   LaserStart_Ext()
   LIN {X 1.720, Y -28.438, Z 22.950}
   LaserEnd_Ext()
   LIN {X 2.720, Y -27.441, Z 22.950}
   LaserStart_Ext()
   LIN {X 2.720, Y 39.118, Z 22.950}
   LaserEnd_Ext()
   LIN {X 3.720, Y 35.905, Z 22.950}
   LaserStart_Ext()
   LIN {X 3.720, Y -25.441, Z 22.950}
   LaserEnd_Ext()
   LIN {X 4.720, Y -22.355, Z 22.950}
   LaserStart_Ext()
   LIN {X 4.720, Y 32.224, Z 22.950}
   LaserEnd_Ext()
   LIN {X 5.720, Y 28.019, Z 22.950}
   LaserStart_Ext()
   LIN {X 5.720, Y -18.121, Z 22.950}
   LaserEnd_Ext()
   LIN {X 6.720, Y -12.774, Z 22.950}
   LaserStart_Ext()
   LIN {X 6.720, Y 22.583, Z 22.950}
   LaserEnd_Ext()
   LIN {X 7.720, Y 14.905, Z 22.950}
   LaserStart_Ext()
   LIN {X 7.720, Y -4.969, Z 22.950}
   LaserEnd_Ext()
   LIN {X -0.569, Y -18.768, Z 23.800}
   LaserStart_Ext()
   LIN {X 0.218, Y -19.359, Z 23.800} C_DIS
   LIN {X 0.697, Y -20.340, Z 23.800} C_DIS
   LIN {X 1.338, Y -21.643, Z 23.800} C_DIS
   LIN {X 1.314, Y -22.747, Z 23.800} C_DIS
   LIN {X 1.286, Y -23.819, Z 23.800} C_DIS
   LIN {X 0.696, Y -24.975, Z 23.800} C_DIS
   LIN {X 0.224, Y -25.880, Z 23.800} C_DIS
   LIN {X -0.464, Y -26.392, Z 23.800} C_DIS
   LIN {X -1.551, Y -27.214, Z 23.800} C_DIS
   LIN {X -3.664, Y -27.649, Z 23.800} C_DIS
   LIN {X -3.922, Y -27.593, Z 23.800} C_DIS
   LIN {X -5.673, Y -27.207, Z 23.800} C_DIS
   LIN {X -7.126, Y -26.129, Z 23.800} C_DIS
   LIN {X -7.331, Y -25.976, Z 23.800} C_DIS
   LIN {X -7.494, Y -25.689, Z 23.800} C_DIS
   LIN {X -8.349, Y -24.188, Z 23.800} C_DIS
   LIN {X -8.499, Y -22.630, Z 23.800} C_DIS
   LIN {X -8.549, Y -22.171, Z 23.800} C_DIS
   LIN {X -8.508, Y -21.998, Z 23.800} C_DIS
   LIN {X -8.307, Y -21.606, Z 23.800} C_DIS
   LIN {X -7.236, Y -19.264, Z 23.800} C_DIS
   LIN {X -5.530, Y -18.053, Z 23.800} C_DIS
   LIN {X -4.970, Y -17.940, Z 23.800} C_DIS
   LIN {X -3.503, Y -17.647, Z 23.800} C_DIS
   LIN {X -2.373, Y -17.894, Z 23.800} C_DIS
   LIN {X -1.482, Y -18.086, Z 23.800} C_DIS
   LIN {X -0.569, Y -18.768, Z 23.800}
   LaserEnd_Ext()
   LIN {X -9.493, Y -14.716, Z 23.800}
   LaserStart_Ext()
   LIN {X -9.270, Y -14.247, Z 23.800} C_DIS
   LIN {X -7.563, Y -10.615, Z 23.800} C_DIS
   LIN {X -6.096, Y -6.905, Z 23.800} C_DIS
   LIN {X -5.884, Y -6.373, Z 23.800} C_DIS
   LIN {X -5.593, Y -5.440, Z 23.800} C_DIS
   LIN {X -4.023, Y -0.432, Z 23.800} C_DIS
   LIN {X -3.188, Y 3.138, Z 23.800} C_DIS
   LIN {X -2.971, Y 4.113, Z 23.800} C_DIS
   LIN {X -2.513, Y 6.884, Z 23.800} C_DIS
   LIN {X -2.208, Y 8.691, Z 23.800} C_DIS
   LIN {X -2.174, Y 8.967, Z 23.800} C_DIS
   LIN {X -1.817, Y 12.348, Z 23.800} C_DIS
   LIN {X -1.729, Y 13.559, Z 23.800} C_DIS
   LIN {X -1.697, Y 15.626, Z 23.800} C_DIS
   LIN {X -1.672, Y 18.321, Z 23.800} C_DIS
   LIN {X -1.649, Y 21.542, Z 23.800} C_DIS
   LIN {X -1.905, Y 24.867, Z 23.800} C_DIS
   LIN {X -2.060, Y 26.694, Z 23.800} C_DIS
   LIN {X -2.450, Y 29.467, Z 23.800} C_DIS
   LIN {X -2.582, Y 30.379, Z 23.800} C_DIS
   LIN {X -3.012, Y 32.709, Z 23.800} C_DIS
   LIN {X -3.518, Y 35.029, Z 23.800} C_DIS
   LIN {X -3.817, Y 36.241, Z 23.800} C_DIS
   LIN {X -3.902, Y 36.583, Z 23.800} C_DIS
   LIN {X -4.015, Y 37.014, Z 23.800} C_DIS
   LIN {X -4.218, Y 37.794, Z 23.800} C_DIS
   LIN {X -4.291, Y 38.488, Z 23.800} C_DIS
   LIN {X -4.358, Y 39.188, Z 23.800} C_DIS
   LIN {X -4.077, Y 40.123, Z 23.800} C_DIS
   LIN {X -3.903, Y 40.742, Z 23.800} C_DIS
   LIN {X -3.579, Y 41.112, Z 23.800} C_DIS
   LIN {X -2.716, Y 42.095, Z 23.800} C_DIS
   LIN {X -0.784, Y 42.721, Z 23.800} C_DIS
   LIN {X -0.398, Y 42.840, Z 23.800} C_DIS
   LIN {X -0.004, Y 42.750, Z 23.800} C_DIS
   LIN {X 1.306, Y 42.455, Z 23.800} C_DIS
   LIN {X 1.975, Y 41.937, Z 23.800} C_DIS
   LIN {X 2.681, Y 41.387, Z 23.800} C_DIS
   LIN {X 3.233, Y 40.398, Z 23.800} C_DIS
   LIN {X 3.399, Y 40.101, Z 23.800} C_DIS
   LIN {X 3.476, Y 39.867, Z 23.800} C_DIS
   LIN {X 3.864, Y 38.690, Z 23.800} C_DIS
   LIN {X 4.445, Y 36.821, Z 23.800} C_DIS
   LIN {X 4.562, Y 36.440, Z 23.800} C_DIS
   LIN {X 4.847, Y 35.435, Z 23.800} C_DIS
   LIN {X 5.308, Y 33.824, Z 23.800} C_DIS
   LIN {X 5.446, Y 33.304, Z 23.800} C_DIS
   LIN {X 6.101, Y 30.733, Z 23.800} C_DIS
   LIN {X 6.906, Y 27.137, Z 23.800} C_DIS
   LIN {X 6.995, Y 26.718, Z 23.800} C_DIS
   LIN {X 7.152, Y 25.799, Z 23.800} C_DIS
   LIN {X 7.886, Y 21.656, Z 23.800} C_DIS
   LIN {X 8.486, Y 16.779, Z 23.800} C_DIS
   LIN {X 8.818, Y 13.934, Z 23.800} C_DIS
   LIN {X 8.922, Y 12.654, Z 23.800} C_DIS
   LIN {X 8.987, Y 11.052, Z 23.800} C_DIS
   LIN {X 9.178, Y 3.666, Z 23.800} C_DIS
   LIN {X 9.014, Y -1.066, Z 23.800} C_DIS
   LIN {X 8.883, Y -3.674, Z 23.800} C_DIS
   LIN {X 8.477, Y -7.663, Z 23.800} C_DIS
   LIN {X 8.257, Y -9.645, Z 23.800} C_DIS
   LIN {X 7.562, Y -14.047, Z 23.800} C_DIS
   LIN {X 7.403, Y -15.079, Z 23.800} C_DIS
   LIN {X 7.324, Y -15.482, Z 23.800} C_DIS
   LIN {X 6.637, Y -18.891, Z 23.800} C_DIS
   LIN {X 6.165, Y -20.922, Z 23.800} C_DIS
   LIN {X 5.938, Y -21.874, Z 23.800} C_DIS
   LIN {X 5.605, Y -23.120, Z 23.800} C_DIS
   LIN {X 5.106, Y -25.030, Z 23.800} C_DIS
   LIN {X 4.234, Y -26.667, Z 23.800} C_DIS
   LIN {X 3.458, Y -28.220, Z 23.800} C_DIS
   LIN {X 2.263, Y -29.368, Z 23.800} C_DIS
   LIN {X 1.337, Y -30.163, Z 23.800} C_DIS
   LIN {X -0.156, Y -30.701, Z 23.800} C_DIS
   LIN {X -2.367, Y -31.568, Z 23.800} C_DIS
   LIN {X -4.741, Y -31.502, Z 23.800} C_DIS
   LIN {X -5.334, Y -31.495, Z 23.800} C_DIS
   LIN {X -5.641, Y -31.410, Z 23.800} C_DIS
   LIN {X -6.673, Y -30.958, Z 23.800} C_DIS
   LIN {X -8.505, Y -30.223, Z 23.800} C_DIS
   LIN {X -9.221, Y -29.523, Z 23.800} C_DIS
   LIN {X -11.153, Y -27.580, Z 23.800} C_DIS
   LIN {X -12.067, Y -25.462, Z 23.800} C_DIS
   LIN {X -12.331, Y -24.860, Z 23.800} C_DIS
   LIN {X -12.375, Y -23.669, Z 23.800} C_DIS
   LIN {X -12.456, Y -21.151, Z 23.800} C_DIS
   LIN {X -12.029, Y -19.995, Z 23.800} C_DIS
   LIN {X -11.371, Y -18.173, Z 23.800} C_DIS
   LIN {X -9.760, Y -15.202, Z 23.800} C_DIS
   LIN {X -9.493, Y -14.716, Z 23.800}
   LaserEnd_Ext()
   LIN {X -2.027, Y -30.360, Z 23.800}
   LaserStart_Ext()
   LIN {X -5.545, Y -30.360, Z 23.800}
   LaserEnd_Ext()
   LIN {X -7.957, Y -29.360, Z 23.800}
   LaserStart_Ext()
   LIN {X 0.616, Y -29.360, Z 23.800}
   LaserEnd_Ext()
   LIN {X 1.868, Y -28.360, Z 23.800}
   LaserStart_Ext()
   LIN {X -2.158, Y -28.360, Z 23.800}
   LaserEnd_Ext()
   LIN {X -5.088, Y -28.360, Z 23.800}
   LaserStart_Ext()
   LIN {X -8.967, Y -28.360, Z 23.800}
   LaserEnd_Ext()
   LIN {X -9.961, Y -27.360, Z 23.800}
   LaserStart_Ext()
   LIN {X -7.145, Y -27.360, Z 23.800}
   LaserEnd_Ext()
   LIN {X -0.087, Y -27.360, Z 23.800}
   LaserStart_Ext()
   LIN {X 2.769, Y -27.360, Z 23.800}
   LaserEnd_Ext()
   LIN {X 3.269, Y -26.360, Z 23.800}
   LaserStart_Ext()
   LIN {X 1.101, Y -26.360, Z 23.800}
   LaserEnd_Ext()
   LIN {X -8.262, Y -26.360, Z 23.800}
   LaserStart_Ext()
   LIN {X -10.590, Y -26.360, Z 23.800}
   LaserEnd_Ext()
   LIN {X -11.021, Y -25.360, Z 23.800}
   LaserStart_Ext()
   LIN {X -8.832, Y -25.360, Z 23.800}
   LaserEnd_Ext()
   LIN {X 1.622, Y -25.360, Z 23.800}
   LaserStart_Ext()
   LIN {X 3.797, Y -25.360, Z 23.800}
   LaserEnd_Ext()
   LIN {X 4.247, Y -24.360, Z 23.800}
   LaserStart_Ext()
   LIN {X 2.133, Y -24.360, Z 23.800}
   LaserEnd_Ext()
   LIN {X -9.333, Y -24.360, Z 23.800}
   LaserStart_Ext()
   LIN {X -11.348, Y -24.360, Z 23.800}
   LaserEnd_Ext()
   LIN {X -11.384, Y -23.360, Z 23.800}
   LaserStart_Ext()
   LIN {X -9.433, Y -23.360, Z 23.800}
   LaserEnd_Ext()
   LIN {X 2.299, Y -23.360, Z 23.800}
   LaserStart_Ext()
   LIN {X 4.508, Y -23.360, Z 23.800}
   LaserEnd_Ext()
   LIN {X 4.773, Y -22.360, Z 23.800}
   LaserStart_Ext()
   LIN {X 2.323, Y -22.360, Z 23.800}
   LaserEnd_Ext()
   LIN {X -9.535, Y -22.360, Z 23.800}
   LaserStart_Ext()
   LIN {X -11.417, Y -22.360, Z 23.800}
   LaserEnd_Ext()
   LIN {X -11.449, Y -21.360, Z 23.800}
   LaserStart_Ext()
   LIN {X -9.305, Y -21.360, Z 23.800}
   LaserEnd_Ext()
   LIN {X 2.297, Y -21.360, Z 23.800}
   LaserStart_Ext()
   LIN {X 5.032, Y -21.360, Z 23.800}
   LaserEnd_Ext()
   LIN {X 5.269, Y -20.360, Z 23.800}
   LaserStart_Ext()
   LIN {X 1.821, Y -20.360, Z 23.800}
   LaserEnd_Ext()
   LIN {X -8.837, Y -20.360, Z 23.800}
   LaserStart_Ext()
   LIN {X -11.098, Y -20.360, Z 23.800}
   LaserEnd_Ext()
   LIN {X -10.737, Y -19.360, Z 23.800}
   LaserStart_Ext()
   LIN {X -8.379, Y -19.360, Z 23.800}
   LaserEnd_Ext()
   LIN {X 1.331, Y -19.360, Z 23.800}
   LaserStart_Ext()
   LIN {X 5.501, Y -19.360, Z 23.800}
   LaserEnd_Ext()
   LIN {X 5.724, Y -18.360, Z 23.800}
   LaserStart_Ext()
   LIN {X 0.553, Y -18.360, Z 23.800}
   LaserEnd_Ext()
   LIN {X -7.690, Y -18.360, Z 23.800}
   LaserStart_Ext()
   LIN {X -10.335, Y -18.360, Z 23.800}
   LaserEnd_Ext()
   LIN {X -9.793, Y -17.360, Z 23.800}
   LaserStart_Ext()
   LIN {X -6.281, Y -17.360, Z 23.800}
   LaserEnd_Ext()
   LIN {X -0.782, Y -17.360, Z 23.800}
   LaserStart_Ext()
   LIN {X 5.925, Y -17.360, Z 23.800}
   LaserEnd_Ext()
   LIN {X 6.127, Y -16.360, Z 23.800}
   LaserStart_Ext()
   LIN {X -9.251, Y -16.360, Z 23.800}
   LaserEnd_Ext()
   LIN {X -8.706, Y -15.360, Z 23.800}
   LaserStart_Ext()
   LIN {X 6.329, Y -15.360, Z 23.800}
   LaserEnd_Ext()
   LIN {X 6.502, Y -14.360, Z 23.800}
   LaserStart_Ext()
   LIN {X -8.218, Y -14.360, Z 23.800}
   LaserEnd_Ext()
   LIN {X -7.748, Y -13.360, Z 23.800}
   LaserStart_Ext()
   LIN {X 6.658, Y -13.360, Z 23.800}
   LaserEnd_Ext()
   LIN {X 6.816, Y -12.360, Z 23.800}
   LaserStart_Ext()
   LIN {X -7.278, Y -12.360, Z 23.800}
   LaserEnd_Ext()
   LIN {X -6.808, Y -11.360, Z 23.800}
   LaserStart_Ext()
   LIN {X 6.974, Y -11.360, Z 23.800}
   LaserEnd_Ext()
   LIN {X 7.132, Y -10.360, Z 23.800}
   LaserStart_Ext()
   LIN {X -6.387, Y -10.360, Z 23.800}
   LaserEnd_Ext()
   LIN {X -5.991, Y -9.360, Z 23.800}
   LaserStart_Ext()
   LIN {X 7.283, Y -9.360, Z 23.800}
   LaserEnd_Ext()
   LIN {X 7.393, Y -8.360, Z 23.800}
   LaserStart_Ext()
   LIN {X -5.596, Y -8.360, Z 23.800}
   LaserEnd_Ext()
   LIN {X -5.201, Y -7.360, Z 23.800}
   LaserStart_Ext()
   LIN {X 7.502, Y -7.360, Z 23.800}
   LaserEnd_Ext()
   LIN {X 7.604, Y -6.360, Z 23.800}
   LaserStart_Ext()
   LIN {X -4.832, Y -6.360, Z 23.800}
   LaserEnd_Ext()
   LIN {X -4.520, Y -5.360, Z 23.800}
   LaserStart_Ext()
   LIN {X 7.706, Y -5.360, Z 23.800}
   LaserEnd_Ext()
   LIN {X 7.808, Y -4.360, Z 23.800}
   LaserStart_Ext()
   LIN {X -4.206, Y -4.360, Z 23.800}
   LaserEnd_Ext()
   LIN {X -3.893, Y -3.360, Z 23.800}
   LaserStart_Ext()
   LIN {X 7.897, Y -3.360, Z 23.800}
   LaserEnd_Ext()
   LIN {X 7.947, Y -2.360, Z 23.800}
   LaserStart_Ext()
   LIN {X -3.580, Y -2.360, Z 23.800}
   LaserEnd_Ext()
   LIN {X -3.266, Y -1.360, Z 23.800}
   LaserStart_Ext()
   LIN {X 7.998, Y -1.360, Z 23.800}
   LaserEnd_Ext()
   LIN {X 8.037, Y -0.360, Z 23.800}
   LaserStart_Ext()
   LIN {X -2.980, Y -0.360, Z 23.800}
   LaserEnd_Ext()
   LIN {X -2.746, Y 0.640, Z 23.800}
   LaserStart_Ext()
   LIN {X 8.072, Y 0.640, Z 23.800}
   LaserEnd_Ext()
   LIN {X 8.107, Y 1.640, Z 23.800}
   LaserStart_Ext()
   LIN {X -2.512, Y 1.640, Z 23.800}
   LaserEnd_Ext()
   LIN {X -2.278, Y 2.640, Z 23.800}
   LaserStart_Ext()
   LIN {X 8.142, Y 2.640, Z 23.800}
   LaserEnd_Ext()
   LIN {X 8.176, Y 3.640, Z 23.800}
   LaserStart_Ext()
   LIN {X -2.052, Y 3.640, Z 23.800}
   LaserEnd_Ext()
   LIN {X -1.870, Y 4.640, Z 23.800}
   LaserStart_Ext()
   LIN {X 8.152, Y 4.640, Z 23.800}
   LaserEnd_Ext()
   LIN {X 8.126, Y 5.640, Z 23.800}
   LaserStart_Ext()
   LIN {X -1.705, Y 5.640, Z 23.800}
   LaserEnd_Ext()
   LIN {X -1.539, Y 6.640, Z 23.800}
   LaserStart_Ext()
   LIN {X 8.101, Y 6.640, Z 23.800}
   LaserEnd_Ext()
   LIN {X 8.075, Y 7.640, Z 23.800}
   LaserStart_Ext()
   LIN {X -1.371, Y 7.640, Z 23.800}
   LaserEnd_Ext()
   LIN {X -1.207, Y 8.640, Z 23.800}
   LaserStart_Ext()
   LIN {X 8.049, Y 8.640, Z 23.800}
   LaserEnd_Ext()
   LIN {X 8.023, Y 9.640, Z 23.800}
   LaserStart_Ext()
   LIN {X -1.097, Y 9.640, Z 23.800}
   LaserEnd_Ext()
   LIN {X -0.992, Y 10.640, Z 23.800}
   LaserStart_Ext()
   LIN {X 7.998, Y 10.640, Z 23.800}
   LaserEnd_Ext()
   LIN {X 7.963, Y 11.640, Z 23.800}
   LaserStart_Ext()
   LIN {X -0.887, Y 11.640, Z 23.800}
   LaserEnd_Ext()
   LIN {X -0.794, Y 12.640, Z 23.800}
   LaserStart_Ext()
   LIN {X 7.920, Y 12.640, Z 23.800}
   LaserEnd_Ext()
   LIN {X 7.839, Y 13.640, Z 23.800}
   LaserStart_Ext()
   LIN {X -0.728, Y 13.640, Z 23.800}
   LaserEnd_Ext()
   LIN {X -0.712, Y 14.640, Z 23.800}
   LaserStart_Ext()
   LIN {X 7.729, Y 14.640, Z 23.800}
   LaserEnd_Ext()
   LIN {X 7.612, Y 15.640, Z 23.800}
   LaserStart_Ext()
   LIN {X -0.696, Y 15.640, Z 23.800}
   LaserEnd_Ext()
   LIN {X -0.687, Y 16.640, Z 23.800}
   LaserStart_Ext()
   LIN {X 7.496, Y 16.640, Z 23.800}
   LaserEnd_Ext()
   LIN {X 7.373, Y 17.640, Z 23.800}
   LaserStart_Ext()
   LIN {X -0.678, Y 17.640, Z 23.800}
   LaserEnd_Ext()
   LIN {X -0.670, Y 18.640, Z 23.800}
   LaserStart_Ext()
   LIN {X 7.250, Y 18.640, Z 23.800}
   LaserEnd_Ext()
   LIN {X 7.126, Y 19.640, Z 23.800}
   LaserStart_Ext()
   LIN {X -0.663, Y 19.640, Z 23.800}
   LaserEnd_Ext()
   LIN {X -0.656, Y 20.640, Z 23.800}
   LaserStart_Ext()
   LIN {X 7.003, Y 20.640, Z 23.800}
   LaserEnd_Ext()
   LIN {X 6.873, Y 21.640, Z 23.800}
   LaserStart_Ext()
   LIN {X -0.654, Y 21.640, Z 23.800}
   LaserEnd_Ext()
   LIN {X -0.731, Y 22.640, Z 23.800}
   LaserStart_Ext()
   LIN {X 6.696, Y 22.640, Z 23.800}
   LaserEnd_Ext()
   LIN {X 6.519, Y 23.640, Z 23.800}
   LaserStart_Ext()
   LIN {X -0.808, Y 23.640, Z 23.800}
   LaserEnd_Ext()
   LIN {X -0.885, Y 24.640, Z 23.800}
   LaserStart_Ext()
   LIN {X 6.342, Y 24.640, Z 23.800}
   LaserEnd_Ext()
   LIN {X 6.165, Y 25.640, Z 23.800}
   LaserStart_Ext()
   LIN {X -0.967, Y 25.640, Z 23.800}
   LaserEnd_Ext()
   LIN {X -1.052, Y 26.640, Z 23.800}
   LaserStart_Ext()
   LIN {X 5.989, Y 26.640, Z 23.800}
   LaserEnd_Ext()
   LIN {X 5.768, Y 27.640, Z 23.800}
   LaserStart_Ext()
   LIN {X -1.183, Y 27.640, Z 23.800}
   LaserEnd_Ext()
   LIN {X -1.324, Y 28.640, Z 23.800}
   LaserStart_Ext()
   LIN {X 5.544, Y 28.640, Z 23.800}
   LaserEnd_Ext()
   LIN {X 5.320, Y 29.640, Z 23.800}
   LaserStart_Ext()
   LIN {X -1.465, Y 29.640, Z 23.800}
   LaserEnd_Ext()
   LIN {X -1.614, Y 30.640, Z 23.800}
   LaserStart_Ext()
   LIN {X 5.092, Y 30.640, Z 23.800}
   LaserEnd_Ext()
   LIN {X 4.838, Y 31.640, Z 23.800}
   LaserStart_Ext()
   LIN {X -1.798, Y 31.640, Z 23.800}
   LaserEnd_Ext()
   LIN {X -1.982, Y 32.640, Z 23.800}
   LaserStart_Ext()
   LIN {X 4.583, Y 32.640, Z 23.800}
   LaserEnd_Ext()
   LIN {X 4.321, Y 33.640, Z 23.800}
   LaserStart_Ext()
   LIN {X -2.192, Y 33.640, Z 23.800}
   LaserEnd_Ext()
   LIN {X -2.410, Y 34.640, Z 23.800}
   LaserStart_Ext()
   LIN {X 4.035, Y 34.640, Z 23.800}
   LaserEnd_Ext()
   LIN {X 3.750, Y 35.640, Z 23.800}
   LaserStart_Ext()
   LIN {X -2.639, Y 35.640, Z 23.800}
   LaserEnd_Ext()
   LIN {X -2.886, Y 36.640, Z 23.800}
   LaserStart_Ext()
   LIN {X 3.454, Y 36.640, Z 23.800}
   LaserEnd_Ext()
   LIN {X 3.143, Y 37.640, Z 23.800}
   LaserStart_Ext()
   LIN {X -3.145, Y 37.640, Z 23.800}
   LaserEnd_Ext()
   LIN {X -3.301, Y 38.640, Z 23.800}
   LaserStart_Ext()
   LIN {X 2.827, Y 38.640, Z 23.800}
   LaserEnd_Ext()
   LIN {X 2.498, Y 39.640, Z 23.800}
   LaserStart_Ext()
   LIN {X -3.178, Y 39.640, Z 23.800}
   LaserEnd_Ext()
   LIN {X -2.663, Y 40.640, Z 23.800}
   LaserStart_Ext()
   LIN {X 1.953, Y 40.640, Z 23.800}
   LaserEnd_Ext()
   LIN {X 0.375, Y 41.640, Z 23.800}
   LaserStart_Ext()
   LIN {X -0.876, Y 41.640, Z 23.800}
   LaserEnd_Ext()
   LIN {X 1.133, Y -24.197, Z 24.650}
   LaserStart_Ext()
   LIN {X 0.254, Y -25.886, Z 24.650} C_DIS
   LIN {X -1.281, Y -27.025, Z 24.650} C_DIS
   LIN {X -1.476, Y -27.168, Z 24.650} C_DIS
   LIN {X -1.626, Y -27.199, Z 24.650} C_DIS
   LIN {X -3.582, Y -27.603, Z 24.650} C_DIS
   LIN {X -5.071, Y -27.279, Z 24.650} C_DIS
   LIN {X -5.588, Y -27.165, Z 24.650} C_DIS
   LIN {X -6.157, Y -26.743, Z 24.650} C_DIS
   LIN {X -7.248, Y -25.938, Z 24.650} C_DIS
   LIN {X -7.835, Y -24.910, Z 24.650} C_DIS
   LIN {X -8.275, Y -24.137, Z 24.650} C_DIS
   LIN {X -8.370, Y -23.158, Z 24.650} C_DIS
   LIN {X -8.472, Y -22.081, Z 24.650} C_DIS
   LIN {X -7.641, Y -20.269, Z 24.650} C_DIS
   LIN {X -7.159, Y -19.216, Z 24.650} C_DIS
   LIN {X -5.458, Y -18.008, Z 24.650} C_DIS
   LIN {X -3.439, Y -17.601, Z 24.650} C_DIS
   LIN {X -3.240, Y -17.643, Z 24.650} C_DIS
   LIN {X -1.418, Y -18.034, Z 24.650} C_DIS
   LIN {X -0.160, Y -18.974, Z 24.650} C_DIS
   LIN {X 0.285, Y -19.304, Z 24.650} C_DIS
   LIN {X 0.602, Y -19.942, Z 24.650} C_DIS
   LIN {X 1.411, Y -21.585, Z 24.650} C_DIS
   LIN {X 1.372, Y -23.366, Z 24.650} C_DIS
   LIN {X 1.364, Y -23.761, Z 24.650} C_DIS
   LIN {X 1.133, Y -24.197, Z 24.650}
   LaserEnd_Ext()
   LIN {X -2.762, Y 31.133, Z 24.650}
   LaserStart_Ext()
   LIN {X -3.068, Y 32.759, Z 24.650} C_DIS
   LIN {X -3.545, Y 34.923, Z 24.650} C_DIS
   LIN {X -3.579, Y 35.075, Z 24.650} C_DIS
   LIN {X -3.622, Y 35.248, Z 24.650} C_DIS
   LIN {X -3.967, Y 36.628, Z 24.650} C_DIS
   LIN {X -4.145, Y 37.309, Z 24.650} C_DIS
   LIN {X -4.285, Y 37.838, Z 24.650} C_DIS
   LIN {X -4.370, Y 38.824, Z 24.650} C_DIS
   LIN {X -4.419, Y 39.337, Z 24.650} C_DIS
   LIN {X -4.283, Y 39.791, Z 24.650} C_DIS
   LIN {X -3.951, Y 40.836, Z 24.650} C_DIS
   LIN {X -3.171, Y 41.741, Z 24.650} C_DIS
   LIN {X -2.861, Y 42.094, Z 24.650} C_DIS
   LIN {X -2.300, Y 42.275, Z 24.650} C_DIS
   LIN {X -0.477, Y 42.894, Z 24.650} C_DIS
   LIN {X 0.607, Y 42.653, Z 24.650} C_DIS
   LIN {X 1.227, Y 42.513, Z 24.650} C_DIS
   LIN {X 1.994, Y 41.919, Z 24.650} C_DIS
   LIN {X 2.605, Y 41.448, Z 24.650} C_DIS
   LIN {X 2.849, Y 41.015, Z 24.650} C_DIS
   LIN {X 3.326, Y 40.164, Z 24.650} C_DIS
   LIN {X 3.760, Y 38.857, Z 24.650} C_DIS
   LIN {X 3.794, Y 38.754, Z 24.650} C_DIS
   LIN {X 4.445, Y 36.677, Z 24.650} C_DIS
   LIN {X 4.876, Y 35.205, Z 24.650} C_DIS
   LIN {X 5.190, Y 34.107, Z 24.650} C_DIS
   LIN {X 5.717, Y 32.116, Z 24.650} C_DIS
   LIN {X 6.024, Y 30.910, Z 24.650} C_DIS
   LIN {X 6.570, Y 28.470, Z 24.650} C_DIS
   LIN {X 6.898, Y 27.034, Z 24.650} C_DIS
   LIN {X 7.027, Y 26.424, Z 24.650} C_DIS
   LIN {X 7.806, Y 22.025, Z 24.650} C_DIS
   LIN {X 8.684, Y 14.898, Z 24.650} C_DIS
   LIN {X 8.861, Y 13.379, Z 24.650} C_DIS
   LIN {X 8.917, Y 12.695, Z 24.650} C_DIS
   LIN {X 8.951, Y 11.840, Z 24.650} C_DIS
   LIN {X 9.185, Y 2.787, Z 24.650} C_DIS
   LIN {X 9.083, Y -0.153, Z 24.650} C_DIS
   LIN {X 8.904, Y -3.715, Z 24.650} C_DIS
   LIN {X 8.349, Y -9.163, Z 24.650} C_DIS
   LIN {X 8.315, Y -9.471, Z 24.650} C_DIS
   LIN {X 8.207, Y -10.154, Z 24.650} C_DIS
   LIN {X 7.461, Y -15.007, Z 24.650} C_DIS
   LIN {X 7.090, Y -16.901, Z 24.650} C_DIS
   LIN {X 6.702, Y -18.821, Z 24.650} C_DIS
   LIN {X 6.053, Y -21.619, Z 24.650} C_DIS
   LIN {X 6.010, Y -21.805, Z 24.650} C_DIS
   LIN {X 5.985, Y -21.906, Z 24.650} C_DIS
   LIN {X 5.186, Y -24.963, Z 24.650} C_DIS
   LIN {X 3.692, Y -27.769, Z 24.650} C_DIS
   LIN {X 3.412, Y -28.329, Z 24.650} C_DIS
   LIN {X 2.982, Y -28.742, Z 24.650} C_DIS
   LIN {X 1.306, Y -30.182, Z 24.650} C_DIS
   LIN {X -1.397, Y -31.154, Z 24.650} C_DIS
   LIN {X -2.354, Y -31.530, Z 24.650} C_DIS
   LIN {X -4.162, Y -31.480, Z 24.650} C_DIS
   LIN {X -5.318, Y -31.437, Z 24.650} C_DIS
   LIN {X -5.693, Y -31.287, Z 24.650} C_DIS
   LIN {X -8.375, Y -30.211, Z 24.650} C_DIS
   LIN {X -10.071, Y -28.553, Z 24.650} C_DIS
   LIN {X -11.066, Y -27.552, Z 24.650} C_DIS
   LIN {X -11.537, Y -26.461, Z 24.650} C_DIS
   LIN {X -12.251, Y -24.834, Z 24.650} C_DIS
   LIN {X -12.370, Y -21.612, Z 24.650} C_DIS
   LIN {X -12.386, Y -21.125, Z 24.650} C_DIS
   LIN {X -12.304, Y -20.902, Z 24.650} C_DIS
   LIN {X -11.307, Y -18.144, Z 24.650} C_DIS
   LIN {X -9.869, Y -15.492, Z 24.650} C_DIS
   LIN {X -9.438, Y -14.685, Z 24.650} C_DIS
   LIN {X -8.973, Y -13.682, Z 24.650} C_DIS
   LIN {X -7.538, Y -10.628, Z 24.650} C_DIS
   LIN {X -6.280, Y -7.446, Z 24.650} C_DIS
   LIN {X -5.878, Y -6.418, Z 24.650} C_DIS
   LIN {X -5.525, Y -5.287, Z 24.650} C_DIS
   LIN {X -4.061, Y -0.614, Z 24.650} C_DIS
   LIN {X -3.469, Y 1.918, Z 24.650} C_DIS
   LIN {X -2.921, Y 4.371, Z 24.650} C_DIS
   LIN {X -2.252, Y 8.420, Z 24.650} C_DIS
   LIN {X -2.236, Y 8.524, Z 24.650} C_DIS
   LIN {X -2.116, Y 9.642, Z 24.650} C_DIS
   LIN {X -1.820, Y 12.450, Z 24.650} C_DIS
   LIN {X -1.762, Y 13.250, Z 24.650} C_DIS
   LIN {X -1.740, Y 14.615, Z 24.650} C_DIS
   LIN {X -1.724, Y 16.395, Z 24.650} C_DIS
   LIN {X -1.686, Y 21.764, Z 24.650} C_DIS
   LIN {X -1.800, Y 23.240, Z 24.650} C_DIS
   LIN {X -2.084, Y 26.596, Z 24.650} C_DIS
   LIN {X -2.331, Y 28.352, Z 24.650} C_DIS
   LIN {X -2.632, Y 30.428, Z 24.650} C_DIS
   LIN {X -2.762, Y 31.133, Z 24.650}
   LaserEnd_Ext()
   LIN {X 7.602, Y -6.629, Z 24.650}
   LaserStart_Ext()
   LIN {X 7.602, Y 15.501, Z 24.650}
   LaserEnd_Ext()
   LIN {X 6.602, Y 23.091, Z 24.650}
   LaserStart_Ext()
   LIN {X 6.602, Y -14.011, Z 24.650}
   LaserEnd_Ext()
   LIN {X 5.602, Y -19.139, Z 24.650}
   LaserStart_Ext()
   LIN {X 5.602, Y 28.220, Z 24.650}
   LaserEnd_Ext()
   LIN {X 4.602, Y 32.421, Z 24.650}
   LaserStart_Ext()
   LIN {X 4.602, Y -23.242, Z 24.650}
   LaserEnd_Ext()
   LIN {X 3.602, Y -25.810, Z 24.650}
   LaserStart_Ext()
   LIN {X 3.602, Y 35.998, Z 24.650}
   LaserEnd_Ext()
   LIN {X 2.602, Y 39.170, Z 24.650}
   LaserStart_Ext()
   LIN {X 2.602, Y -27.713, Z 24.650}
   LaserEnd_Ext()
   LIN {X 1.602, Y -28.609, Z 24.650}
   LaserStart_Ext()
   LIN {X 1.602, Y -25.462, Z 24.650}
   LaserEnd_Ext()
   LIN {X 1.602, Y -19.709, Z 24.650}
   LaserStart_Ext()
   LIN {X 1.602, Y 40.959, Z 24.650}
   LaserEnd_Ext()
   LIN {X 0.602, Y 41.629, Z 24.650}
   LaserStart_Ext()
   LIN {X 0.602, Y -18.294, Z 24.650}
   LaserEnd_Ext()
   LIN {X 0.602, Y -26.873, Z 24.650}
   LaserStart_Ext()
   LIN {X 0.602, Y -29.372, Z 24.650}
   LaserEnd_Ext()
   LIN {X -0.398, Y -29.732, Z 24.650}
   LaserStart_Ext()
   LIN {X -0.398, Y -27.615, Z 24.650}
   LaserEnd_Ext()
   LIN {X -0.398, Y -17.548, Z 24.650}
   LaserStart_Ext()
   LIN {X -0.398, Y 41.852, Z 24.650}
   LaserEnd_Ext()
   LIN {X -1.398, Y 41.525, Z 24.650}
   LaserStart_Ext()
   LIN {X -1.398, Y 28.888, Z 24.650}
   LaserEnd_Ext()
   LIN {X -1.398, Y 7.454, Z 24.650}
   LaserStart_Ext()
   LIN {X -1.398, Y -17.016, Z 24.650}
   LaserEnd_Ext()
   LIN {X -1.398, Y -28.173, Z 24.650}
   LaserStart_Ext()
   LIN {X -1.398, Y -30.092, Z 24.650}
   LaserEnd_Ext()
   LIN {X -2.398, Y -30.473, Z 24.650}
   LaserStart_Ext()
   LIN {X -2.398, Y -28.380, Z 24.650}
   LaserEnd_Ext()
   LIN {X -2.398, Y -16.801, Z 24.650}
   LaserStart_Ext()
   LIN {X -2.398, Y 2.124, Z 24.650}
   LaserEnd_Ext()
   LIN {X -2.398, Y 34.365, Z 24.650}
   LaserStart_Ext()
   LIN {X -2.398, Y 41.105, Z 24.650}
   LaserEnd_Ext()
   LIN {X -3.398, Y 39.261, Z 24.650}
   LaserStart_Ext()
   LIN {X -3.398, Y 39.163, Z 24.650}
   LaserEnd_Ext()
   LIN {X -3.398, Y -1.843, Z 24.650}
   LaserStart_Ext()
   LIN {X -3.398, Y -16.603, Z 24.650}
   LaserEnd_Ext()
   LIN {X -3.398, Y -28.585, Z 24.650}
   LaserStart_Ext()
   LIN {X -3.398, Y -30.501, Z 24.650}
   LaserEnd_Ext()
   LIN {X -4.398, Y -30.470, Z 24.650}
   LaserStart_Ext()
   LIN {X -4.398, Y -28.449, Z 24.650}
   LaserEnd_Ext()
   LIN {X -4.398, Y -16.774, Z 24.650}
   LaserStart_Ext()
   LIN {X -4.398, Y -5.034, Z 24.650}
   LaserEnd_Ext()
   LIN {X -5.398, Y -7.935, Z 24.650}
   LaserStart_Ext()
   LIN {X -5.398, Y -16.976, Z 24.650}
   LaserEnd_Ext()
   LIN {X -5.398, Y -28.231, Z 24.650}
   LaserStart_Ext()
   LIN {X -5.398, Y -30.328, Z 24.650}
   LaserEnd_Ext()
   LIN {X -6.398, Y -29.927, Z 24.650}
   LaserStart_Ext()
   LIN {X -6.398, Y -27.809, Z 24.650}
   LaserEnd_Ext()
   LIN {X -6.398, Y -17.449, Z 24.650}
   LaserStart_Ext()
   LIN {X -6.398, Y -10.465, Z 24.650}
   LaserEnd_Ext()
   LIN {X -7.398, Y -12.681, Z 24.650}
   LaserStart_Ext()
   LIN {X -7.398, Y -18.159, Z 24.650}
   LaserEnd_Ext()
   LIN {X -7.398, Y -27.070, Z 24.650}
   LaserStart_Ext()
   LIN {X -7.398, Y -29.526, Z 24.650}
   LaserEnd_Ext()
   LIN {X -8.398, Y -28.790, Z 24.650}
   LaserStart_Ext()
   LIN {X -8.398, Y -25.941, Z 24.650}
   LaserEnd_Ext()
   LIN {X -8.398, Y -19.520, Z 24.650}
   LaserStart_Ext()
   LIN {X -8.398, Y -14.819, Z 24.650}
   LaserEnd_Ext()
   LIN {X -9.398, Y -16.721, Z 24.650}
   LaserStart_Ext()
   LIN {X -9.398, Y -21.708, Z 24.650}
   LaserEnd_Ext()
   LIN {X -9.398, Y -22.905, Z 24.650}
   LaserStart_Ext()
   LIN {X -9.398, Y -27.812, Z 24.650}
   LaserEnd_Ext()
   LIN {X -10.398, Y -26.577, Z 24.650}
   LaserStart_Ext()
   LIN {X -10.398, Y -18.573, Z 24.650}
   LaserEnd_Ext()
   LIN {X 0.353, Y -19.248, Z 25.500}
   LaserStart_Ext()
   LIN {X 1.449, Y -21.457, Z 25.500} C_DIS
   LIN {X 1.482, Y -21.602, Z 25.500} C_DIS
   LIN {X 1.442, Y -23.702, Z 25.500} C_DIS
   LIN {X 0.338, Y -25.789, Z 25.500} C_DIS
   LIN {X 0.287, Y -25.888, Z 25.500} C_DIS
   LIN {X -1.401, Y -27.121, Z 25.500} C_DIS
   LIN {X -2.793, Y -27.410, Z 25.500} C_DIS
   LIN {X -3.499, Y -27.556, Z 25.500} C_DIS
   LIN {X -4.487, Y -27.342, Z 25.500} C_DIS
   LIN {X -5.502, Y -27.124, Z 25.500} C_DIS
   LIN {X -6.151, Y -26.649, Z 25.500} C_DIS
   LIN {X -7.165, Y -25.900, Z 25.500} C_DIS
   LIN {X -7.887, Y -24.637, Z 25.500} C_DIS
   LIN {X -8.200, Y -24.092, Z 25.500} C_DIS
   LIN {X -8.257, Y -23.498, Z 25.500} C_DIS
   LIN {X -8.396, Y -22.030, Z 25.500} C_DIS
   LIN {X -7.588, Y -20.267, Z 25.500} C_DIS
   LIN {X -7.083, Y -19.168, Z 25.500} C_DIS
   LIN {X -5.385, Y -17.962, Z 25.500} C_DIS
   LIN {X -3.366, Y -17.554, Z 25.500} C_DIS
   LIN {X -1.592, Y -17.932, Z 25.500} C_DIS
   LIN {X -1.353, Y -17.983, Z 25.500} C_DIS
   LIN {X -1.189, Y -18.106, Z 25.500} C_DIS
   LIN {X 0.353, Y -19.248, Z 25.500}
   LaserEnd_Ext()
   LIN {X 4.519, Y 36.260, Z 25.500}
   LaserStart_Ext()
   LIN {X 5.040, Y 34.496, Z 25.500} C_DIS
   LIN {X 5.173, Y 34.026, Z 25.500} C_DIS
   LIN {X 5.940, Y 31.117, Z 25.500} C_DIS
   LIN {X 5.969, Y 31.001, Z 25.500} C_DIS
   LIN {X 6.760, Y 27.534, Z 25.500} C_DIS
   LIN {X 7.108, Y 25.887, Z 25.500} C_DIS
   LIN {X 7.727, Y 22.394, Z 25.500} C_DIS
   LIN {X 8.881, Y 13.017, Z 25.500} C_DIS
   LIN {X 8.904, Y 12.823, Z 25.500} C_DIS
   LIN {X 8.915, Y 12.627, Z 25.500} C_DIS
   LIN {X 9.192, Y 1.908, Z 25.500} C_DIS
   LIN {X 9.152, Y 0.760, Z 25.500} C_DIS
   LIN {X 8.925, Y -3.755, Z 25.500} C_DIS
   LIN {X 8.860, Y -4.394, Z 25.500} C_DIS
   LIN {X 8.351, Y -9.472, Z 25.500} C_DIS
   LIN {X 8.115, Y -11.056, Z 25.500} C_DIS
   LIN {X 7.518, Y -14.934, Z 25.500} C_DIS
   LIN {X 6.855, Y -18.321, Z 25.500} C_DIS
   LIN {X 6.768, Y -18.750, Z 25.500} C_DIS
   LIN {X 6.623, Y -19.376, Z 25.500} C_DIS
   LIN {X 6.084, Y -21.736, Z 25.500} C_DIS
   LIN {X 5.759, Y -23.009, Z 25.500} C_DIS
   LIN {X 5.266, Y -24.895, Z 25.500} C_DIS
   LIN {X 3.815, Y -27.621, Z 25.500} C_DIS
   LIN {X 3.476, Y -28.295, Z 25.500} C_DIS
   LIN {X 3.126, Y -28.610, Z 25.500} C_DIS
   LIN {X 1.275, Y -30.200, Z 25.500} C_DIS
   LIN {X -2.109, Y -31.418, Z 25.500} C_DIS
   LIN {X -2.338, Y -31.491, Z 25.500} C_DIS
   LIN {X -2.560, Y -31.479, Z 25.500} C_DIS
   LIN {X -5.302, Y -31.378, Z 25.500} C_DIS
   LIN {X -6.442, Y -30.923, Z 25.500} C_DIS
   LIN {X -8.246, Y -30.199, Z 25.500} C_DIS
   LIN {X -10.922, Y -27.584, Z 25.500} C_DIS
   LIN {X -11.008, Y -27.461, Z 25.500} C_DIS
   LIN {X -12.171, Y -24.808, Z 25.500} C_DIS
   LIN {X -12.278, Y -21.910, Z 25.500} C_DIS
   LIN {X -12.315, Y -21.099, Z 25.500} C_DIS
   LIN {X -11.905, Y -19.948, Z 25.500} C_DIS
   LIN {X -11.243, Y -18.116, Z 25.500} C_DIS
   LIN {X -10.455, Y -16.663, Z 25.500} C_DIS
   LIN {X -9.386, Y -14.662, Z 25.500} C_DIS
   LIN {X -8.235, Y -12.177, Z 25.500} C_DIS
   LIN {X -7.513, Y -10.641, Z 25.500} C_DIS
   LIN {X -6.880, Y -9.041, Z 25.500} C_DIS
   LIN {X -5.859, Y -6.429, Z 25.500} C_DIS
   LIN {X -4.963, Y -3.554, Z 25.500} C_DIS
   LIN {X -4.099, Y -0.796, Z 25.500} C_DIS
   LIN {X -3.749, Y 0.698, Z 25.500} C_DIS
   LIN {X -2.871, Y 4.628, Z 25.500} C_DIS
   LIN {X -2.335, Y 7.875, Z 25.500} C_DIS
   LIN {X -2.292, Y 8.155, Z 25.500} C_DIS
   LIN {X -1.967, Y 11.189, Z 25.500} C_DIS
   LIN {X -1.823, Y 12.553, Z 25.500} C_DIS
   LIN {X -1.795, Y 12.941, Z 25.500} C_DIS
   LIN {X -1.784, Y 13.604, Z 25.500} C_DIS
   LIN {X -1.776, Y 14.468, Z 25.500} C_DIS
   LIN {X -1.735, Y 20.306, Z 25.500} C_DIS
   LIN {X -1.720, Y 21.921, Z 25.500} C_DIS
   LIN {X -1.804, Y 22.916, Z 25.500} C_DIS
   LIN {X -2.108, Y 26.498, Z 25.500} C_DIS
   LIN {X -2.211, Y 27.236, Z 25.500} C_DIS
   LIN {X -2.422, Y 28.687, Z 25.500} C_DIS
   LIN {X -2.682, Y 30.476, Z 25.500} C_DIS
   LIN {X -3.002, Y 32.163, Z 25.500} C_DIS
   LIN {X -3.123, Y 32.807, Z 25.500} C_DIS
   LIN {X -3.208, Y 33.191, Z 25.500} C_DIS
   LIN {X -3.640, Y 35.121, Z 25.500} C_DIS
   LIN {X -3.945, Y 36.334, Z 25.500} C_DIS
   LIN {X -4.031, Y 36.673, Z 25.500} C_DIS
   LIN {X -4.172, Y 37.201, Z 25.500} C_DIS
   LIN {X -4.353, Y 37.883, Z 25.500} C_DIS
   LIN {X -4.401, Y 38.444, Z 25.500} C_DIS
   LIN {X -4.485, Y 39.434, Z 25.500} C_DIS
   LIN {X -4.134, Y 40.517, Z 25.500} C_DIS
   LIN {X -4.009, Y 40.912, Z 25.500} C_DIS
   LIN {X -3.733, Y 41.231, Z 25.500} C_DIS
   LIN {X -2.936, Y 42.144, Z 25.500} C_DIS
   LIN {X -0.851, Y 42.847, Z 25.500} C_DIS
   LIN {X -0.556, Y 42.947, Z 25.500} C_DIS
   LIN {X -0.278, Y 42.885, Z 25.500} C_DIS
   LIN {X 1.149, Y 42.570, Z 25.500} C_DIS
   LIN {X 1.751, Y 42.109, Z 25.500} C_DIS
   LIN {X 2.529, Y 41.508, Z 25.500} C_DIS
   LIN {X 3.051, Y 40.582, Z 25.500} C_DIS
   LIN {X 3.253, Y 40.226, Z 25.500} C_DIS
   LIN {X 3.357, Y 39.916, Z 25.500} C_DIS
   LIN {X 3.724, Y 38.817, Z 25.500} C_DIS
   LIN {X 4.232, Y 37.220, Z 25.500} C_DIS
   LIN {X 4.315, Y 36.956, Z 25.500} C_DIS
   LIN {X 4.519, Y 36.260, Z 25.500}
   LaserEnd_Ext()
   LIN {X -1.652, Y 41.522, Z 25.500}
   LaserStart_Ext()
   LIN {X 0.873, Y 41.522, Z 25.500}
   LaserEnd_Ext()
   LIN {X 1.937, Y 40.522, Z 25.500}
   LaserStart_Ext()
   LIN {X -3.025, Y 40.522, Z 25.500}
   LaserEnd_Ext()
   LIN {X -3.405, Y 39.522, Z 25.500}
   LaserStart_Ext()
   LIN {X 2.435, Y 39.522, Z 25.500}
   LaserEnd_Ext()
   LIN {X 2.769, Y 38.522, Z 25.500}
   LaserStart_Ext()
   LIN {X -3.404, Y 38.522, Z 25.500}
   LaserEnd_Ext()
   LIN {X -3.222, Y 37.522, Z 25.500}
   LaserStart_Ext()
   LIN {X 3.087, Y 37.522, Z 25.500}
   LaserEnd_Ext()
   LIN {X 3.400, Y 36.522, Z 25.500}
   LaserStart_Ext()
   LIN {X -2.961, Y 36.522, Z 25.500}
   LaserEnd_Ext()
   LIN {X -2.710, Y 35.522, Z 25.500}
   LaserStart_Ext()
   LIN {X 3.694, Y 35.522, Z 25.500}
   LaserEnd_Ext()
   LIN {X 3.990, Y 34.522, Z 25.500}
   LaserStart_Ext()
   LIN {X -2.481, Y 34.522, Z 25.500}
   LaserEnd_Ext()
   LIN {X -2.257, Y 33.522, Z 25.500}
   LaserStart_Ext()
   LIN {X 4.272, Y 33.522, Z 25.500}
   LaserEnd_Ext()
   LIN {X 4.535, Y 32.522, Z 25.500}
   LaserStart_Ext()
   LIN {X -2.052, Y 32.522, Z 25.500}
   LaserEnd_Ext()
   LIN {X -1.863, Y 31.522, Z 25.500}
   LaserStart_Ext()
   LIN {X 4.799, Y 31.522, Z 25.500}
   LaserEnd_Ext()
   LIN {X 5.052, Y 30.522, Z 25.500}
   LaserStart_Ext()
   LIN {X -1.678, Y 30.522, Z 25.500}
   LaserEnd_Ext()
   LIN {X -1.533, Y 29.522, Z 25.500}
   LaserStart_Ext()
   LIN {X 5.281, Y 29.522, Z 25.500}
   LaserEnd_Ext()
   LIN {X 5.509, Y 28.522, Z 25.500}
   LaserStart_Ext()
   LIN {X -1.388, Y 28.522, Z 25.500}
   LaserEnd_Ext()
   LIN {X -1.242, Y 27.522, Z 25.500}
   LaserStart_Ext()
   LIN {X 5.737, Y 27.522, Z 25.500}
   LaserEnd_Ext()
   LIN {X 5.952, Y 26.522, Z 25.500}
   LaserStart_Ext()
   LIN {X -1.106, Y 26.522, Z 25.500}
   LaserEnd_Ext()
   LIN {X -1.021, Y 25.522, Z 25.500}
   LaserStart_Ext()
   LIN {X 6.157, Y 25.522, Z 25.500}
   LaserEnd_Ext()
   LIN {X 6.334, Y 24.522, Z 25.500}
   LaserStart_Ext()
   LIN {X -0.937, Y 24.522, Z 25.500}
   LaserEnd_Ext()
   LIN {X -0.852, Y 23.522, Z 25.500}
   LaserStart_Ext()
   LIN {X 6.512, Y 23.522, Z 25.500}
   LaserEnd_Ext()
   LIN {X 6.689, Y 22.522, Z 25.500}
   LaserStart_Ext()
   LIN {X -0.767, Y 22.522, Z 25.500}
   LaserEnd_Ext()
   LIN {X -0.723, Y 21.522, Z 25.500}
   LaserStart_Ext()
   LIN {X 6.827, Y 21.522, Z 25.500}
   LaserEnd_Ext()
   LIN {X 6.950, Y 20.522, Z 25.500}
   LaserStart_Ext()
   LIN {X -0.733, Y 20.522, Z 25.500}
   LaserEnd_Ext()
   LIN {X -0.740, Y 19.522, Z 25.500}
   LaserStart_Ext()
   LIN {X 7.073, Y 19.522, Z 25.500}
   LaserEnd_Ext()
   LIN {X 7.196, Y 18.522, Z 25.500}
   LaserStart_Ext()
   LIN {X -0.748, Y 18.522, Z 25.500}
   LaserEnd_Ext()
   LIN {X -0.755, Y 17.522, Z 25.500}
   LaserStart_Ext()
   LIN {X 7.319, Y 17.522, Z 25.500}
   LaserEnd_Ext()
   LIN {X 7.442, Y 16.522, Z 25.500}
   LaserStart_Ext()
   LIN {X -0.762, Y 16.522, Z 25.500}
   LaserEnd_Ext()
   LIN {X -0.769, Y 15.522, Z 25.500}
   LaserStart_Ext()
   LIN {X 7.565, Y 15.522, Z 25.500}
   LaserEnd_Ext()
   LIN {X 7.688, Y 14.522, Z 25.500}
   LaserStart_Ext()
   LIN {X -0.776, Y 14.522, Z 25.500}
   LaserEnd_Ext()
   LIN {X -0.785, Y 13.522, Z 25.500}
   LaserStart_Ext()
   LIN {X 7.812, Y 13.522, Z 25.500}
   LaserEnd_Ext()
   LIN {X 7.918, Y 12.522, Z 25.500}
   LaserStart_Ext()
   LIN {X -0.823, Y 12.522, Z 25.500}
   LaserEnd_Ext()
   LIN {X -0.926, Y 11.522, Z 25.500}
   LaserStart_Ext()
   LIN {X 7.943, Y 11.522, Z 25.500}
   LaserEnd_Ext()
   LIN {X 7.969, Y 10.522, Z 25.500}
   LaserStart_Ext()
   LIN {X -1.032, Y 10.522, Z 25.500}
   LaserEnd_Ext()
   LIN {X -1.140, Y 9.522, Z 25.500}
   LaserStart_Ext()
   LIN {X 7.995, Y 9.522, Z 25.500}
   LaserEnd_Ext()
   LIN {X 8.021, Y 8.522, Z 25.500}
   LaserStart_Ext()
   LIN {X -1.247, Y 8.522, Z 25.500}
   LaserEnd_Ext()
   LIN {X -1.380, Y 7.522, Z 25.500}
   LaserStart_Ext()
   LIN {X 8.047, Y 7.522, Z 25.500}
   LaserEnd_Ext()
   LIN {X 8.072, Y 6.522, Z 25.500}
   LaserStart_Ext()
   LIN {X -1.545, Y 6.522, Z 25.500}
   LaserEnd_Ext()
   LIN {X -1.710, Y 5.522, Z 25.500}
   LaserStart_Ext()
   LIN {X 8.098, Y 5.522, Z 25.500}
   LaserEnd_Ext()
   LIN {X 8.124, Y 4.522, Z 25.500}
   LaserStart_Ext()
   LIN {X -1.876, Y 4.522, Z 25.500}
   LaserEnd_Ext()
   LIN {X -2.094, Y 3.522, Z 25.500}
   LaserStart_Ext()
   LIN {X 8.150, Y 3.522, Z 25.500}
   LaserEnd_Ext()
   LIN {X 8.176, Y 2.522, Z 25.500}
   LaserStart_Ext()
   LIN {X -2.317, Y 2.522, Z 25.500}
   LaserEnd_Ext()
   LIN {X -2.541, Y 1.522, Z 25.500}
   LaserStart_Ext()
   LIN {X 8.178, Y 1.522, Z 25.500}
   LaserEnd_Ext()
   LIN {X 8.139, Y 0.522, Z 25.500}
   LaserStart_Ext()
   LIN {X -2.764, Y 0.522, Z 25.500}
   LaserEnd_Ext()
   LIN {X -2.997, Y -0.478, Z 25.500}
   LaserStart_Ext()
   LIN {X 8.088, Y -0.478, Z 25.500}
   LaserEnd_Ext()
   LIN {X 8.038, Y -1.478, Z 25.500}
   LaserStart_Ext()
   LIN {X -3.264, Y -1.478, Z 25.500}
   LaserEnd_Ext()
   LIN {X -3.578, Y -2.478, Z 25.500}
   LaserStart_Ext()
   LIN {X 7.988, Y -2.478, Z 25.500}
   LaserEnd_Ext()
   LIN {X 7.938, Y -3.478, Z 25.500}
   LaserStart_Ext()
   LIN {X -3.891, Y -3.478, Z 25.500}
   LaserEnd_Ext()
   LIN {X -4.203, Y -4.478, Z 25.500}
   LaserStart_Ext()
   LIN {X 7.846, Y -4.478, Z 25.500}
   LaserEnd_Ext()
   LIN {X 7.746, Y -5.478, Z 25.500}
   LaserStart_Ext()
   LIN {X -4.515, Y -5.478, Z 25.500}
   LaserEnd_Ext()
   LIN {X -4.827, Y -6.478, Z 25.500}
   LaserStart_Ext()
   LIN {X 7.646, Y -6.478, Z 25.500}
   LaserEnd_Ext()
   LIN {X 7.546, Y -7.478, Z 25.500}
   LaserStart_Ext()
   LIN {X -5.195, Y -7.478, Z 25.500}
   LaserEnd_Ext()
   LIN {X -5.587, Y -8.478, Z 25.500}
   LaserStart_Ext()
   LIN {X 7.445, Y -8.478, Z 25.500}
   LaserEnd_Ext()
   LIN {X 7.339, Y -9.478, Z 25.500}
   LaserStart_Ext()
   LIN {X -5.978, Y -9.478, Z 25.500}
   LaserEnd_Ext()
   LIN {X -6.374, Y -10.478, Z 25.500}
   LaserStart_Ext()
   LIN {X 7.190, Y -10.478, Z 25.500}
   LaserEnd_Ext()
   LIN {X 7.038, Y -11.478, Z 25.500}
   LaserStart_Ext()
   LIN {X -6.802, Y -11.478, Z 25.500}
   LaserEnd_Ext()
   LIN {X -7.272, Y -12.478, Z 25.500}
   LaserStart_Ext()
   LIN {X 6.884, Y -12.478, Z 25.500}
   LaserEnd_Ext()
   LIN {X 6.730, Y -13.478, Z 25.500}
   LaserStart_Ext()
   LIN {X -7.736, Y -13.478, Z 25.500}
   LaserEnd_Ext()
   LIN {X -8.199, Y -14.478, Z 25.500}
   LaserStart_Ext()
   LIN {X 6.576, Y -14.478, Z 25.500}
   LaserEnd_Ext()
   LIN {X 6.392, Y -15.478, Z 25.500}
   LaserStart_Ext()
   LIN {X -8.689, Y -15.478, Z 25.500}
   LaserEnd_Ext()
   LIN {X -9.223, Y -16.478, Z 25.500}
   LaserStart_Ext()
   LIN {X 6.197, Y -16.478, Z 25.500}
   LaserEnd_Ext()
   LIN {X 6.001, Y -17.478, Z 25.500}
   LaserStart_Ext()
   LIN {X -0.356, Y -17.478, Z 25.500}
   LaserEnd_Ext()
   LIN {X -6.431, Y -17.478, Z 25.500}
   LaserStart_Ext()
   LIN {X -9.760, Y -17.478, Z 25.500}
   LaserEnd_Ext()
   LIN {X -10.302, Y -18.478, Z 25.500}
   LaserStart_Ext()
   LIN {X -7.806, Y -18.478, Z 25.500}
   LaserEnd_Ext()
   LIN {X 0.989, Y -18.478, Z 25.500}
   LaserStart_Ext()
   LIN {X 5.803, Y -18.478, Z 25.500}
   LaserEnd_Ext()
   LIN {X 5.574, Y -19.478, Z 25.500}
   LaserStart_Ext()
   LIN {X 1.583, Y -19.478, Z 25.500}
   LaserEnd_Ext()
   LIN {X -8.326, Y -19.478, Z 25.500}
   LaserStart_Ext()
   LIN {X -10.672, Y -19.478, Z 25.500}
   LaserEnd_Ext()
   LIN {X -11.032, Y -20.478, Z 25.500}
   LaserStart_Ext()
   LIN {X -8.785, Y -20.478, Z 25.500}
   LaserEnd_Ext()
   LIN {X 2.080, Y -20.478, Z 25.500}
   LaserStart_Ext()
   LIN {X 5.345, Y -20.478, Z 25.500}
   LaserEnd_Ext()
   LIN {X 5.117, Y -21.478, Z 25.500}
   LaserStart_Ext()
   LIN {X 2.481, Y -21.478, Z 25.500}
   LaserEnd_Ext()
   LIN {X -9.243, Y -21.478, Z 25.500}
   LaserStart_Ext()
   LIN {X -11.297, Y -21.478, Z 25.500}
   LaserEnd_Ext()
   LIN {X -11.257, Y -22.478, Z 25.500}
   LaserStart_Ext()
   LIN {X -9.358, Y -22.478, Z 25.500}
   LaserEnd_Ext()
   LIN {X 2.465, Y -22.478, Z 25.500}
   LaserStart_Ext()
   LIN {X 4.862, Y -22.478, Z 25.500}
   LaserEnd_Ext()
   LIN {X 4.603, Y -23.478, Z 25.500}
   LaserStart_Ext()
   LIN {X 2.446, Y -23.478, Z 25.500}
   LaserEnd_Ext()
   LIN {X -9.263, Y -23.478, Z 25.500}
   LaserStart_Ext()
   LIN {X -11.219, Y -23.478, Z 25.500}
   LaserEnd_Ext()
   LIN {X -11.182, Y -24.478, Z 25.500}
   LaserStart_Ext()
   LIN {X -9.121, Y -24.478, Z 25.500}
   LaserEnd_Ext()
   LIN {X 2.163, Y -24.478, Z 25.500}
   LaserStart_Ext()
   LIN {X 4.342, Y -24.478, Z 25.500}
   LaserEnd_Ext()
   LIN {X 3.823, Y -25.478, Z 25.500}
   LaserStart_Ext()
   LIN {X 1.634, Y -25.478, Z 25.500}
   LaserEnd_Ext()
   LIN {X -8.558, Y -25.478, Z 25.500}
   LaserStart_Ext()
   LIN {X -10.785, Y -25.478, Z 25.500}
   LaserEnd_Ext()
   LIN {X -10.347, Y -26.478, Z 25.500}
   LaserStart_Ext()
   LIN {X -7.981, Y -26.478, Z 25.500}
   LaserEnd_Ext()
   LIN {X 1.092, Y -26.478, Z 25.500}
   LaserStart_Ext()
   LIN {X 3.291, Y -26.478, Z 25.500}
   LaserEnd_Ext()
   LIN {X 2.767, Y -27.478, Z 25.500}
   LaserStart_Ext()
   LIN {X -0.195, Y -27.478, Z 25.500}
   LaserEnd_Ext()
   LIN {X -6.710, Y -27.478, Z 25.500}
   LaserStart_Ext()
   LIN {X -9.599, Y -27.478, Z 25.500}
   LaserEnd_Ext()
   LIN {X -8.575, Y -28.478, Z 25.500}
   LaserStart_Ext()
   LIN {X -3.966, Y -28.478, Z 25.500}
   LaserEnd_Ext()
   LIN {X -3.020, Y -28.478, Z 25.500}
   LaserStart_Ext()
   LIN {X 1.745, Y -28.478, Z 25.500}
   LaserEnd_Ext()
   LIN {X 0.328, Y -29.478, Z 25.500}
   LaserStart_Ext()
   LIN {X -7.356, Y -29.478, Z 25.500}
   LaserEnd_Ext()
   LIN {X -2.567, Y -30.478, Z 25.500}
   LaserStart_Ext()
   LIN {X -2.453, Y -30.478, Z 25.500}
   LaserEnd_Ext()
   LIN {X -5.416, Y -27.082, Z 26.350}
   LaserStart_Ext()
   LIN {X -6.962, Y -25.950, Z 26.350} C_DIS
   LIN {X -7.082, Y -25.862, Z 26.350} C_DIS
   LIN {X -7.147, Y -25.750, Z 26.350} C_DIS
   LIN {X -8.121, Y -24.057, Z 26.350} C_DIS
   LIN {X -8.318, Y -22.008, Z 26.350} C_DIS
   LIN {X -7.006, Y -19.120, Z 26.350} C_DIS
   LIN {X -5.313, Y -17.917, Z 26.350} C_DIS
   LIN {X -3.293, Y -17.507, Z 26.350} C_DIS
   LIN {X -2.376, Y -17.702, Z 26.350} C_DIS
   LIN {X -1.289, Y -17.931, Z 26.350} C_DIS
   LIN {X -0.154, Y -18.767, Z 26.350} C_DIS
   LIN {X 0.420, Y -19.193, Z 26.350} C_DIS
   LIN {X 0.772, Y -19.901, Z 26.350} C_DIS
   LIN {X 1.556, Y -21.468, Z 26.350} C_DIS
   LIN {X 1.536, Y -22.801, Z 26.350} C_DIS
   LIN {X 1.520, Y -23.644, Z 26.350} C_DIS
   LIN {X 1.104, Y -24.430, Z 26.350} C_DIS
   LIN {X 0.362, Y -25.841, Z 26.350} C_DIS
   LIN {X -1.326, Y -27.075, Z 26.350} C_DIS
   LIN {X -2.568, Y -27.333, Z 26.350} C_DIS
   LIN {X -3.415, Y -27.510, Z 26.350} C_DIS
   LIN {X -3.972, Y -27.392, Z 26.350} C_DIS
   LIN {X -5.416, Y -27.082, Z 26.350}
   LaserEnd_Ext()
   LIN {X -4.501, Y 38.908, Z 26.350}
   LaserStart_Ext()
   LIN {X -4.552, Y 39.509, Z 26.350} C_DIS
   LIN {X -4.394, Y 39.999, Z 26.350} C_DIS
   LIN {X -4.068, Y 40.985, Z 26.350} C_DIS
   LIN {X -3.239, Y 41.923, Z 26.350} C_DIS
   LIN {X -2.986, Y 42.212, Z 26.350} C_DIS
   LIN {X -2.503, Y 42.375, Z 26.350} C_DIS
   LIN {X -0.635, Y 43.000, Z 26.350} C_DIS
   LIN {X 0.549, Y 42.742, Z 26.350} C_DIS
   LIN {X 1.071, Y 42.627, Z 26.350} C_DIS
   LIN {X 1.842, Y 42.036, Z 26.350} C_DIS
   LIN {X 2.453, Y 41.569, Z 26.350} C_DIS
   LIN {X 2.659, Y 41.208, Z 26.350} C_DIS
   LIN {X 3.180, Y 40.288, Z 26.350} C_DIS
   LIN {X 3.618, Y 38.988, Z 26.350} C_DIS
   LIN {X 3.655, Y 38.880, Z 26.350} C_DIS
   LIN {X 4.162, Y 37.298, Z 26.350} C_DIS
   LIN {X 4.471, Y 36.295, Z 26.350} C_DIS
   LIN {X 4.843, Y 35.037, Z 26.350} C_DIS
   LIN {X 5.297, Y 33.431, Z 26.350} C_DIS
   LIN {X 5.796, Y 31.539, Z 26.350} C_DIS
   LIN {X 6.073, Y 30.439, Z 26.350} C_DIS
   LIN {X 6.621, Y 28.035, Z 26.350} C_DIS
   LIN {X 7.189, Y 25.350, Z 26.350} C_DIS
   LIN {X 7.647, Y 22.763, Z 26.350} C_DIS
   LIN {X 8.567, Y 15.293, Z 26.350} C_DIS
   LIN {X 8.876, Y 13.062, Z 26.350} C_DIS
   LIN {X 8.920, Y 12.643, Z 26.350} C_DIS
   LIN {X 8.947, Y 12.058, Z 26.350} C_DIS
   LIN {X 9.203, Y 1.442, Z 26.350} C_DIS
   LIN {X 9.194, Y 1.117, Z 26.350} C_DIS
   LIN {X 9.183, Y 0.901, Z 26.350} C_DIS
   LIN {X 8.948, Y -3.796, Z 26.350} C_DIS
   LIN {X 8.804, Y -5.300, Z 26.350} C_DIS
   LIN {X 8.381, Y -9.514, Z 26.350} C_DIS
   LIN {X 7.856, Y -13.038, Z 26.350} C_DIS
   LIN {X 7.575, Y -14.862, Z 26.350} C_DIS
   LIN {X 7.160, Y -16.980, Z 26.350} C_DIS
   LIN {X 6.835, Y -18.679, Z 26.350} C_DIS
   LIN {X 6.670, Y -19.424, Z 26.350} C_DIS
   LIN {X 6.157, Y -21.667, Z 26.350} C_DIS
   LIN {X 5.534, Y -24.112, Z 26.350} C_DIS
   LIN {X 5.347, Y -24.828, Z 26.350} C_DIS
   LIN {X 4.796, Y -25.862, Z 26.350} C_DIS
   LIN {X 3.681, Y -28.079, Z 26.350} C_DIS
   LIN {X 2.531, Y -29.113, Z 26.350} C_DIS
   LIN {X 1.244, Y -30.219, Z 26.350} C_DIS
   LIN {X -1.109, Y -31.066, Z 26.350} C_DIS
   LIN {X -2.310, Y -31.450, Z 26.350} C_DIS
   LIN {X -3.473, Y -31.386, Z 26.350} C_DIS
   LIN {X -5.285, Y -31.319, Z 26.350} C_DIS
   LIN {X -7.191, Y -30.558, Z 26.350} C_DIS
   LIN {X -8.116, Y -30.187, Z 26.350} C_DIS
   LIN {X -9.564, Y -28.772, Z 26.350} C_DIS
   LIN {X -10.893, Y -27.496, Z 26.350} C_DIS
   LIN {X -11.321, Y -26.538, Z 26.350} C_DIS
   LIN {X -12.091, Y -24.781, Z 26.350} C_DIS
   LIN {X -12.159, Y -22.951, Z 26.350} C_DIS
   LIN {X -12.243, Y -21.074, Z 26.350} C_DIS
   LIN {X -11.294, Y -18.407, Z 26.350} C_DIS
   LIN {X -11.179, Y -18.088, Z 26.350} C_DIS
   LIN {X -11.041, Y -17.834, Z 26.350} C_DIS
   LIN {X -9.335, Y -14.640, Z 26.350} C_DIS
   LIN {X -7.497, Y -10.673, Z 26.350} C_DIS
   LIN {X -5.840, Y -6.440, Z 26.350} C_DIS
   LIN {X -4.400, Y -1.820, Z 26.350} C_DIS
   LIN {X -4.136, Y -0.978, Z 26.350} C_DIS
   LIN {X -4.030, Y -0.522, Z 26.350} C_DIS
   LIN {X -2.822, Y 4.886, Z 26.350} C_DIS
   LIN {X -2.418, Y 7.329, Z 26.350} C_DIS
   LIN {X -2.348, Y 7.786, Z 26.350} C_DIS
   LIN {X -1.832, Y 12.597, Z 26.350} C_DIS
   LIN {X -1.825, Y 12.828, Z 26.350} C_DIS
   LIN {X -1.741, Y 21.823, Z 26.350} C_DIS
   LIN {X -2.095, Y 25.981, Z 26.350} C_DIS
   LIN {X -2.135, Y 26.432, Z 26.350} C_DIS
   LIN {X -2.169, Y 26.660, Z 26.350} C_DIS
   LIN {X -2.198, Y 26.852, Z 26.350} C_DIS
   LIN {X -2.389, Y 28.166, Z 26.350} C_DIS
   LIN {X -2.732, Y 30.524, Z 26.350} C_DIS
   LIN {X -2.875, Y 31.278, Z 26.350} C_DIS
   LIN {X -3.179, Y 32.854, Z 26.350} C_DIS
   LIN {X -3.626, Y 34.831, Z 26.350} C_DIS
   LIN {X -3.701, Y 35.167, Z 26.350} C_DIS
   LIN {X -3.737, Y 35.310, Z 26.350} C_DIS
   LIN {X -4.096, Y 36.718, Z 26.350} C_DIS
   LIN {X -4.291, Y 37.449, Z 26.350} C_DIS
   LIN {X -4.420, Y 37.927, Z 26.350} C_DIS
   LIN {X -4.501, Y 38.908, Z 26.350}
   LaserEnd_Ext()
   LIN {X -10.280, Y -18.543, Z 26.350}
   LaserStart_Ext()
   LIN {X -10.280, Y -26.416, Z 26.350}
   LaserEnd_Ext()
   LIN {X -9.280, Y -27.658, Z 26.350}
   LaserStart_Ext()
   LIN {X -9.280, Y -22.454, Z 26.350}
   LaserEnd_Ext()
   LIN {X -9.280, Y -21.701, Z 26.350}
   LaserStart_Ext()
   LIN {X -9.280, Y -16.659, Z 26.350}
   LaserEnd_Ext()
   LIN {X -8.280, Y -14.742, Z 26.350}
   LaserStart_Ext()
   LIN {X -8.280, Y -19.496, Z 26.350}
   LaserEnd_Ext()
   LIN {X -8.280, Y -25.787, Z 26.350}
   LaserStart_Ext()
   LIN {X -8.280, Y -28.629, Z 26.350}
   LaserEnd_Ext()
   LIN {X -7.280, Y -29.445, Z 26.350}
   LaserStart_Ext()
   LIN {X -7.280, Y -26.956, Z 26.350}
   LaserEnd_Ext()
   LIN {X -7.280, Y -18.087, Z 26.350}
   LaserStart_Ext()
   LIN {X -7.280, Y -12.583, Z 26.350}
   LaserEnd_Ext()
   LIN {X -6.280, Y -10.310, Z 26.350}
   LaserStart_Ext()
   LIN {X -6.280, Y -17.377, Z 26.350}
   LaserEnd_Ext()
   LIN {X -6.280, Y -27.689, Z 26.350}
   LaserStart_Ext()
   LIN {X -6.280, Y -29.845, Z 26.350}
   LaserEnd_Ext()
   LIN {X -5.280, Y -30.245, Z 26.350}
   LaserStart_Ext()
   LIN {X -5.280, Y -28.134, Z 26.350}
   LaserEnd_Ext()
   LIN {X -5.280, Y -16.890, Z 26.350}
   LaserStart_Ext()
   LIN {X -5.280, Y -7.754, Z 26.350}
   LaserEnd_Ext()
   LIN {X -4.280, Y -4.796, Z 26.350}
   LaserStart_Ext()
   LIN {X -4.280, Y -16.687, Z 26.350}
   LaserEnd_Ext()
   LIN {X -4.280, Y -28.349, Z 26.350}
   LaserStart_Ext()
   LIN {X -4.280, Y -30.356, Z 26.350}
   LaserEnd_Ext()
   LIN {X -3.280, Y -30.395, Z 26.350}
   LaserStart_Ext()
   LIN {X -3.280, Y -28.499, Z 26.350}
   LaserEnd_Ext()
   LIN {X -3.280, Y -16.508, Z 26.350}
   LaserStart_Ext()
   LIN {X -3.280, Y -1.590, Z 26.350}
   LaserEnd_Ext()
   LIN {X -3.280, Y 37.539, Z 26.350}
   LaserStart_Ext()
   LIN {X -3.280, Y 40.182, Z 26.350}
   LaserEnd_Ext()
   LIN {X -2.280, Y 41.395, Z 26.350}
   LaserStart_Ext()
   LIN {X -2.280, Y 33.412, Z 26.350}
   LaserEnd_Ext()
   LIN {X -2.280, Y 2.725, Z 26.350}
   LaserStart_Ext()
   LIN {X -2.280, Y -16.700, Z 26.350}
   LaserEnd_Ext()
   LIN {X -2.280, Y -28.294, Z 26.350}
   LaserStart_Ext()
   LIN {X -2.280, Y -30.390, Z 26.350}
   LaserEnd_Ext()
   LIN {X -1.280, Y -30.064, Z 26.350}
   LaserStart_Ext()
   LIN {X -1.280, Y -28.087, Z 26.350}
   LaserEnd_Ext()
   LIN {X -1.280, Y -16.911, Z 26.350}
   LaserStart_Ext()
   LIN {X -1.280, Y 8.371, Z 26.350}
   LaserEnd_Ext()
   LIN {X -1.280, Y 27.489, Z 26.350}
   LaserStart_Ext()
   LIN {X -1.280, Y 41.730, Z 26.350}
   LaserEnd_Ext()
   LIN {X -0.280, Y 41.899, Z 26.350}
   LaserStart_Ext()
   LIN {X -0.280, Y -17.432, Z 26.350}
   LaserEnd_Ext()
   LIN {X -0.280, Y -27.549, Z 26.350}
   LaserStart_Ext()
   LIN {X -0.280, Y -29.705, Z 26.350}
   LaserEnd_Ext()
   LIN {X 0.720, Y -29.345, Z 26.350}
   LaserStart_Ext()
   LIN {X 0.720, Y -26.818, Z 26.350}
   LaserEnd_Ext()
   LIN {X 0.720, Y -18.171, Z 26.350}
   LaserStart_Ext()
   LIN {X 0.720, Y 41.636, Z 26.350}
   LaserEnd_Ext()
   LIN {X 1.720, Y 40.836, Z 26.350}
   LaserStart_Ext()
   LIN {X 1.720, Y -19.562, Z 26.350}
   LaserEnd_Ext()
   LIN {X 1.720, Y -25.407, Z 26.350}
   LaserStart_Ext()
   LIN {X 1.720, Y -28.491, Z 26.350}
   LaserEnd_Ext()
   LIN {X 2.720, Y -27.598, Z 26.350}
   LaserStart_Ext()
   LIN {X 2.720, Y 38.521, Z 26.350}
   LaserEnd_Ext()
   LIN {X 3.720, Y 35.307, Z 26.350}
   LaserStart_Ext()
   LIN {X 3.720, Y -25.776, Z 26.350}
   LaserEnd_Ext()
   LIN {X 4.720, Y -23.255, Z 26.350}
   LaserStart_Ext()
   LIN {X 4.720, Y 31.697, Z 26.350}
   LaserEnd_Ext()
   LIN {X 5.720, Y 27.462, Z 26.350}
   LaserStart_Ext()
   LIN {X 5.720, Y -19.087, Z 26.350}
   LaserEnd_Ext()
   LIN {X 6.720, Y -13.843, Z 26.350}
   LaserStart_Ext()
   LIN {X 6.720, Y 22.110, Z 26.350}
   LaserEnd_Ext()
   LIN {X 7.720, Y 14.118, Z 26.350}
   LaserStart_Ext()
   LIN {X 7.720, Y -6.083, Z 26.350}
   LaserEnd_Ext()
   LIN {X 1.629, Y -21.410, Z 27.200}
   LaserStart_Ext()
   LIN {X 1.606, Y -22.911, Z 27.200} C_DIS
   LIN {X 1.598, Y -23.586, Z 27.200} C_DIS
   LIN {X 1.170, Y -24.402, Z 27.200} C_DIS
   LIN {X 0.437, Y -25.794, Z 27.200} C_DIS
   LIN {X -0.659, Y -26.596, Z 27.200} C_DIS
   LIN {X -1.247, Y -27.026, Z 27.200} C_DIS
   LIN {X -1.712, Y -27.125, Z 27.200} C_DIS
   LIN {X -3.328, Y -27.463, Z 27.200} C_DIS
   LIN {X -5.166, Y -27.075, Z 27.200} C_DIS
   LIN {X -5.330, Y -27.040, Z 27.200} C_DIS
   LIN {X -5.506, Y -26.911, Z 27.200} C_DIS
   LIN {X -6.999, Y -25.824, Z 27.200} C_DIS
   LIN {X -7.807, Y -24.431, Z 27.200} C_DIS
   LIN {X -8.043, Y -24.021, Z 27.200} C_DIS
   LIN {X -8.090, Y -23.526, Z 27.200} C_DIS
   LIN {X -8.247, Y -21.945, Z 27.200} C_DIS
   LIN {X -7.198, Y -19.655, Z 27.200} C_DIS
   LIN {X -6.930, Y -19.072, Z 27.200} C_DIS
   LIN {X -5.239, Y -17.870, Z 27.200} C_DIS
   LIN {X -3.562, Y -17.530, Z 27.200} C_DIS
   LIN {X -3.234, Y -17.460, Z 27.200} C_DIS
   LIN {X -2.771, Y -17.554, Z 27.200} C_DIS
   LIN {X -1.225, Y -17.879, Z 27.200} C_DIS
   LIN {X -0.139, Y -18.679, Z 27.200} C_DIS
   LIN {X 0.488, Y -19.137, Z 27.200} C_DIS
   LIN {X 0.938, Y -20.029, Z 27.200} C_DIS
   LIN {X 1.629, Y -21.410, Z 27.200}
   LaserEnd_Ext()
   LIN {X -0.109, Y -30.713, Z 27.200}
   LaserStart_Ext()
   LIN {X 1.213, Y -30.237, Z 27.200} C_DIS
   LIN {X 1.936, Y -29.616, Z 27.200} C_DIS
   LIN {X 3.886, Y -27.863, Z 27.200} C_DIS
   LIN {X 5.226, Y -25.198, Z 27.200} C_DIS
   LIN {X 5.427, Y -24.760, Z 27.200} C_DIS
   LIN {X 5.628, Y -23.961, Z 27.200} C_DIS
   LIN {X 6.231, Y -21.597, Z 27.200} C_DIS
   LIN {X 6.505, Y -20.399, Z 27.200} C_DIS
   LIN {X 6.901, Y -18.608, Z 27.200} C_DIS
   LIN {X 7.600, Y -14.962, Z 27.200} C_DIS
   LIN {X 7.632, Y -14.789, Z 27.200} C_DIS
   LIN {X 7.683, Y -14.440, Z 27.200} C_DIS
   LIN {X 8.412, Y -9.555, Z 27.200} C_DIS
   LIN {X 8.666, Y -7.016, Z 27.200} C_DIS
   LIN {X 8.972, Y -3.837, Z 27.200} C_DIS
   LIN {X 9.147, Y -0.332, Z 27.200} C_DIS
   LIN {X 9.189, Y 0.482, Z 27.200} C_DIS
   LIN {X 9.220, Y 1.713, Z 27.200} C_DIS
   LIN {X 8.991, Y 11.256, Z 27.200} C_DIS
   LIN {X 8.931, Y 12.527, Z 27.200} C_DIS
   LIN {X 8.836, Y 13.436, Z 27.200} C_DIS
   LIN {X 8.165, Y 18.280, Z 27.200} C_DIS
   LIN {X 7.568, Y 23.132, Z 27.200} C_DIS
   LIN {X 7.270, Y 24.812, Z 27.200} C_DIS
   LIN {X 6.483, Y 28.535, Z 27.200} C_DIS
   LIN {X 6.177, Y 29.877, Z 27.200} C_DIS
   LIN {X 5.652, Y 31.961, Z 27.200} C_DIS
   LIN {X 5.422, Y 32.836, Z 27.200} C_DIS
   LIN {X 4.738, Y 35.251, Z 27.200} C_DIS
   LIN {X 4.671, Y 35.490, Z 27.200} C_DIS
   LIN {X 4.569, Y 35.819, Z 27.200} C_DIS
   LIN {X 4.004, Y 37.653, Z 27.200} C_DIS
   LIN {X 3.820, Y 38.225, Z 27.200} C_DIS
   LIN {X 3.585, Y 38.943, Z 27.200} C_DIS
   LIN {X 3.193, Y 40.097, Z 27.200} C_DIS
   LIN {X 3.107, Y 40.350, Z 27.200} C_DIS
   LIN {X 2.924, Y 40.669, Z 27.200} C_DIS
   LIN {X 2.378, Y 41.629, Z 27.200} C_DIS
   LIN {X 1.682, Y 42.160, Z 27.200} C_DIS
   LIN {X 0.992, Y 42.684, Z 27.200} C_DIS
   LIN {X -0.144, Y 42.929, Z 27.200} C_DIS
   LIN {X -0.715, Y 43.053, Z 27.200} C_DIS
   LIN {X -1.377, Y 42.831, Z 27.200} C_DIS
   LIN {X -3.072, Y 42.253, Z 27.200} C_DIS
   LIN {X -3.801, Y 41.426, Z 27.200} C_DIS
   LIN {X -4.127, Y 41.056, Z 27.200} C_DIS
   LIN {X -4.295, Y 40.548, Z 27.200} C_DIS
   LIN {X -4.622, Y 39.564, Z 27.200} C_DIS
   LIN {X -4.553, Y 38.766, Z 27.200} C_DIS
   LIN {X -4.487, Y 37.971, Z 27.200} C_DIS
   LIN {X -4.204, Y 36.925, Z 27.200} C_DIS
   LIN {X -4.160, Y 36.763, Z 27.200} C_DIS
   LIN {X -4.127, Y 36.634, Z 27.200} C_DIS
   LIN {X -3.762, Y 35.213, Z 27.200} C_DIS
   LIN {X -3.314, Y 33.255, Z 27.200} C_DIS
   LIN {X -3.234, Y 32.901, Z 27.200} C_DIS
   LIN {X -3.144, Y 32.434, Z 27.200} C_DIS
   LIN {X -2.767, Y 30.487, Z 27.200} C_DIS
   LIN {X -2.463, Y 28.406, Z 27.200} C_DIS
   LIN {X -2.332, Y 27.513, Z 27.200} C_DIS
   LIN {X -2.171, Y 26.454, Z 27.200} C_DIS
   LIN {X -1.986, Y 24.353, Z 27.200} C_DIS
   LIN {X -1.762, Y 21.725, Z 27.200} C_DIS
   LIN {X -1.815, Y 16.038, Z 27.200} C_DIS
   LIN {X -1.836, Y 12.645, Z 27.200} C_DIS
   LIN {X -1.950, Y 11.657, Z 27.200} C_DIS
   LIN {X -2.405, Y 7.417, Z 27.200} C_DIS
   LIN {X -2.501, Y 6.784, Z 27.200} C_DIS
   LIN {X -2.772, Y 5.144, Z 27.200} C_DIS
   LIN {X -3.834, Y 0.390, Z 27.200} C_DIS
   LIN {X -4.173, Y -1.161, Z 27.200} C_DIS
   LIN {X -4.512, Y -2.253, Z 27.200} C_DIS
   LIN {X -5.821, Y -6.451, Z 27.200} C_DIS
   LIN {X -6.921, Y -9.263, Z 27.200} C_DIS
   LIN {X -7.462, Y -10.668, Z 27.200} C_DIS
   LIN {X -8.154, Y -12.179, Z 27.200} C_DIS
   LIN {X -9.283, Y -14.618, Z 27.200} C_DIS
   LIN {X -10.506, Y -16.906, Z 27.200} C_DIS
   LIN {X -11.114, Y -18.059, Z 27.200} C_DIS
   LIN {X -11.360, Y -18.768, Z 27.200} C_DIS
   LIN {X -12.171, Y -21.048, Z 27.200} C_DIS
   LIN {X -12.039, Y -23.991, Z 27.200} C_DIS
   LIN {X -12.011, Y -24.755, Z 27.200} C_DIS
   LIN {X -11.689, Y -25.488, Z 27.200} C_DIS
   LIN {X -10.806, Y -27.467, Z 27.200} C_DIS
   LIN {X -8.059, Y -30.104, Z 27.200} C_DIS
   LIN {X -7.987, Y -30.175, Z 27.200} C_DIS
   LIN {X -5.269, Y -31.260, Z 27.200} C_DIS
   LIN {X -4.387, Y -31.293, Z 27.200} C_DIS
   LIN {X -2.282, Y -31.408, Z 27.200} C_DIS
   LIN {X -0.109, Y -30.713, Z 27.200}
   LaserEnd_Ext()
   LIN {X -2.287, Y -30.360, Z 27.200}
   LaserStart_Ext()
   LIN {X -3.134, Y -30.360, Z 27.200}
   LaserEnd_Ext()
   LIN {X -7.330, Y -29.360, Z 27.200}
   LaserStart_Ext()
   LIN {X 0.698, Y -29.360, Z 27.200}
   LaserEnd_Ext()
   LIN {X 1.837, Y -28.360, Z 27.200}
   LaserStart_Ext()
   LIN {X -2.733, Y -28.360, Z 27.200}
   LaserEnd_Ext()
   LIN {X -3.919, Y -28.360, Z 27.200}
   LaserStart_Ext()
   LIN {X -8.431, Y -28.360, Z 27.200}
   LaserEnd_Ext()
   LIN {X -9.473, Y -27.360, Z 27.200}
   LaserStart_Ext()
   LIN {X -6.588, Y -27.360, Z 27.200}
   LaserEnd_Ext()
   LIN {X -0.011, Y -27.360, Z 27.200}
   LaserStart_Ext()
   LIN {X 2.949, Y -27.360, Z 27.200}
   LaserEnd_Ext()
   LIN {X 3.522, Y -26.360, Z 27.200}
   LaserStart_Ext()
   LIN {X 1.260, Y -26.360, Z 27.200}
   LaserEnd_Ext()
   LIN {X -7.842, Y -26.360, Z 27.200}
   LaserStart_Ext()
   LIN {X -10.205, Y -26.360, Z 27.200}
   LaserEnd_Ext()
   LIN {X -10.651, Y -25.360, Z 27.200}
   LaserStart_Ext()
   LIN {X -8.424, Y -25.360, Z 27.200}
   LaserEnd_Ext()
   LIN {X 1.795, Y -25.360, Z 27.200}
   LaserStart_Ext()
   LIN {X 4.025, Y -25.360, Z 27.200}
   LaserEnd_Ext()
   LIN {X 4.497, Y -24.360, Z 27.200}
   LaserStart_Ext()
   LIN {X 2.321, Y -24.360, Z 27.200}
   LaserEnd_Ext()
   LIN {X -8.982, Y -24.360, Z 27.200}
   LaserStart_Ext()
   LIN {X -11.025, Y -24.360, Z 27.200}
   LaserEnd_Ext()
   LIN {X -11.066, Y -23.360, Z 27.200}
   LaserStart_Ext()
   LIN {X -9.111, Y -23.360, Z 27.200}
   LaserEnd_Ext()
   LIN {X 2.601, Y -23.360, Z 27.200}
   LaserStart_Ext()
   LIN {X 4.749, Y -23.360, Z 27.200}
   LaserEnd_Ext()
   LIN {X 5.004, Y -22.360, Z 27.200}
   LaserStart_Ext()
   LIN {X 2.615, Y -22.360, Z 27.200}
   LaserEnd_Ext()
   LIN {X -9.211, Y -22.360, Z 27.200}
   LaserStart_Ext()
   LIN {X -11.111, Y -22.360, Z 27.200}
   LaserEnd_Ext()
   LIN {X -11.156, Y -21.360, Z 27.200}
   LaserStart_Ext()
   LIN {X -9.079, Y -21.360, Z 27.200}
   LaserEnd_Ext()
   LIN {X 2.627, Y -21.360, Z 27.200}
   LaserStart_Ext()
   LIN {X 5.259, Y -21.360, Z 27.200}
   LaserEnd_Ext()
   LIN {X 5.488, Y -20.360, Z 27.200}
   LaserStart_Ext()
   LIN {X 2.222, Y -20.360, Z 27.200}
   LaserEnd_Ext()
   LIN {X -8.621, Y -20.360, Z 27.200}
   LaserStart_Ext()
   LIN {X -10.865, Y -20.360, Z 27.200}
   LaserEnd_Ext()
   LIN {X -10.509, Y -19.360, Z 27.200}
   LaserStart_Ext()
   LIN {X -8.163, Y -19.360, Z 27.200}
   LaserEnd_Ext()
   LIN {X 1.720, Y -19.360, Z 27.200}
   LaserStart_Ext()
   LIN {X 5.710, Y -19.360, Z 27.200}
   LaserEnd_Ext()
   LIN {X 5.931, Y -18.360, Z 27.200}
   LaserStart_Ext()
   LIN {X 1.115, Y -18.360, Z 27.200}
   LaserEnd_Ext()
   LIN {X -7.631, Y -18.360, Z 27.200}
   LaserStart_Ext()
   LIN {X -10.142, Y -18.360, Z 27.200}
   LaserEnd_Ext()
   LIN {X -9.615, Y -17.360, Z 27.200}
   LaserStart_Ext()
   LIN {X -6.248, Y -17.360, Z 27.200}
   LaserEnd_Ext()
   LIN {X -0.243, Y -17.360, Z 27.200}
   LaserStart_Ext()
   LIN {X 6.122, Y -17.360, Z 27.200}
   LaserEnd_Ext()
   LIN {X 6.314, Y -16.360, Z 27.200}
   LaserStart_Ext()
   LIN {X -9.080, Y -16.360, Z 27.200}
   LaserEnd_Ext()
   LIN {X -8.546, Y -15.360, Z 27.200}
   LaserStart_Ext()
   LIN {X 6.506, Y -15.360, Z 27.200}
   LaserEnd_Ext()
   LIN {X 6.684, Y -14.360, Z 27.200}
   LaserStart_Ext()
   LIN {X -8.062, Y -14.360, Z 27.200}
   LaserEnd_Ext()
   LIN {X -7.599, Y -13.360, Z 27.200}
   LaserStart_Ext()
   LIN {X 6.833, Y -13.360, Z 27.200}
   LaserEnd_Ext()
   LIN {X 6.982, Y -12.360, Z 27.200}
   LaserStart_Ext()
   LIN {X -7.137, Y -12.360, Z 27.200}
   LaserEnd_Ext()
   LIN {X -6.679, Y -11.360, Z 27.200}
   LaserStart_Ext()
   LIN {X 7.131, Y -11.360, Z 27.200}
   LaserEnd_Ext()
   LIN {X 7.281, Y -10.360, Z 27.200}
   LaserStart_Ext()
   LIN {X -6.272, Y -10.360, Z 27.200}
   LaserEnd_Ext()
   LIN {X -5.885, Y -9.360, Z 27.200}
   LaserStart_Ext()
   LIN {X 7.426, Y -9.360, Z 27.200}
   LaserEnd_Ext()
   LIN {X 7.526, Y -8.360, Z 27.200}
   LaserStart_Ext()
   LIN {X -5.494, Y -8.360, Z 27.200}
   LaserEnd_Ext()
   LIN {X -5.102, Y -7.360, Z 27.200}
   LaserStart_Ext()
   LIN {X 7.627, Y -7.360, Z 27.200}
   LaserEnd_Ext()
   LIN {X 7.725, Y -6.360, Z 27.200}
   LaserStart_Ext()
   LIN {X -4.745, Y -6.360, Z 27.200}
   LaserEnd_Ext()
   LIN {X -4.433, Y -5.360, Z 27.200}
   LaserStart_Ext()
   LIN {X 7.821, Y -5.360, Z 27.200}
   LaserEnd_Ext()
   LIN {X 7.917, Y -4.360, Z 27.200}
   LaserStart_Ext()
   LIN {X -4.122, Y -4.360, Z 27.200}
   LaserEnd_Ext()
   LIN {X -3.810, Y -3.360, Z 27.200}
   LaserStart_Ext()
   LIN {X 7.994, Y -3.360, Z 27.200}
   LaserEnd_Ext()
   LIN {X 8.044, Y -2.360, Z 27.200}
   LaserStart_Ext()
   LIN {X -3.498, Y -2.360, Z 27.200}
   LaserEnd_Ext()
   LIN {X -3.193, Y -1.360, Z 27.200}
   LaserStart_Ext()
   LIN {X 8.094, Y -1.360, Z 27.200}
   LaserEnd_Ext()
   LIN {X 8.144, Y -0.360, Z 27.200}
   LaserStart_Ext()
   LIN {X -2.974, Y -0.360, Z 27.200}
   LaserEnd_Ext()
   LIN {X -2.753, Y 0.640, Z 27.200}
   LaserStart_Ext()
   LIN {X 8.193, Y 0.640, Z 27.200}
   LaserEnd_Ext()
   LIN {X 8.218, Y 1.640, Z 27.200}
   LaserStart_Ext()
   LIN {X -2.530, Y 1.640, Z 27.200}
   LaserEnd_Ext()
   LIN {X -2.307, Y 2.640, Z 27.200}
   LaserStart_Ext()
   LIN {X 8.198, Y 2.640, Z 27.200}
   LaserEnd_Ext()
   LIN {X 8.174, Y 3.640, Z 27.200}
   LaserStart_Ext()
   LIN {X -2.084, Y 3.640, Z 27.200}
   LaserEnd_Ext()
   LIN {X -1.860, Y 4.640, Z 27.200}
   LaserStart_Ext()
   LIN {X 8.150, Y 4.640, Z 27.200}
   LaserEnd_Ext()
   LIN {X 8.126, Y 5.640, Z 27.200}
   LaserStart_Ext()
   LIN {X -1.677, Y 5.640, Z 27.200}
   LaserEnd_Ext()
   LIN {X -1.512, Y 6.640, Z 27.200}
   LaserStart_Ext()
   LIN {X 8.102, Y 6.640, Z 27.200}
   LaserEnd_Ext()
   LIN {X 8.078, Y 7.640, Z 27.200}
   LaserStart_Ext()
   LIN {X -1.375, Y 7.640, Z 27.200}
   LaserEnd_Ext()
   LIN {X -1.268, Y 8.640, Z 27.200}
   LaserStart_Ext()
   LIN {X 8.054, Y 8.640, Z 27.200}
   LaserEnd_Ext()
   LIN {X 8.030, Y 9.640, Z 27.200}
   LaserStart_Ext()
   LIN {X -1.160, Y 9.640, Z 27.200}
   LaserEnd_Ext()
   LIN {X -1.053, Y 10.640, Z 27.200}
   LaserStart_Ext()
   LIN {X 8.006, Y 10.640, Z 27.200}
   LaserEnd_Ext()
   LIN {X 7.972, Y 11.640, Z 27.200}
   LaserStart_Ext()
   LIN {X -0.945, Y 11.640, Z 27.200}
   LaserEnd_Ext()
   LIN {X -0.836, Y 12.640, Z 27.200}
   LaserStart_Ext()
   LIN {X 7.914, Y 12.640, Z 27.200}
   LaserEnd_Ext()
   LIN {X 7.798, Y 13.640, Z 27.200}
   LaserStart_Ext()
   LIN {X -0.830, Y 13.640, Z 27.200}
   LaserEnd_Ext()
   LIN {X -0.824, Y 14.640, Z 27.200}
   LaserStart_Ext()
   LIN {X 7.660, Y 14.640, Z 27.200}
   LaserEnd_Ext()
   LIN {X 7.521, Y 15.640, Z 27.200}
   LaserStart_Ext()
   LIN {X -0.817, Y 15.640, Z 27.200}
   LaserEnd_Ext()
   LIN {X -0.809, Y 16.640, Z 27.200}
   LaserStart_Ext()
   LIN {X 7.383, Y 16.640, Z 27.200}
   LaserEnd_Ext()
   LIN {X 7.244, Y 17.640, Z 27.200}
   LaserStart_Ext()
   LIN {X -0.800, Y 17.640, Z 27.200}
   LaserEnd_Ext()
   LIN {X -0.791, Y 18.640, Z 27.200}
   LaserStart_Ext()
   LIN {X 7.113, Y 18.640, Z 27.200}
   LaserEnd_Ext()
   LIN {X 6.990, Y 19.640, Z 27.200}
   LaserStart_Ext()
   LIN {X -0.781, Y 19.640, Z 27.200}
   LaserEnd_Ext()
   LIN {X -0.772, Y 20.640, Z 27.200}
   LaserStart_Ext()
   LIN {X 6.867, Y 20.640, Z 27.200}
   LaserEnd_Ext()
   LIN {X 6.744, Y 21.640, Z 27.200}
   LaserStart_Ext()
   LIN {X -0.763, Y 21.640, Z 27.200}
   LaserEnd_Ext()
   LIN {X -0.836, Y 22.640, Z 27.200}
   LaserStart_Ext()
   LIN {X 6.621, Y 22.640, Z 27.200}
   LaserEnd_Ext()
   LIN {X 6.462, Y 23.640, Z 27.200}
   LaserStart_Ext()
   LIN {X -0.921, Y 23.640, Z 27.200}
   LaserEnd_Ext()
   LIN {X -1.007, Y 24.640, Z 27.200}
   LaserStart_Ext()
   LIN {X 6.285, Y 24.640, Z 27.200}
   LaserEnd_Ext()
   LIN {X 6.073, Y 25.640, Z 27.200}
   LaserStart_Ext()
   LIN {X -1.096, Y 25.640, Z 27.200}
   LaserEnd_Ext()
   LIN {X -1.188, Y 26.640, Z 27.200}
   LaserStart_Ext()
   LIN {X 5.862, Y 26.640, Z 27.200}
   LaserEnd_Ext()
   LIN {X 5.650, Y 27.640, Z 27.200}
   LaserStart_Ext()
   LIN {X -1.340, Y 27.640, Z 27.200}
   LaserEnd_Ext()
   LIN {X -1.486, Y 28.640, Z 27.200}
   LaserStart_Ext()
   LIN {X 5.433, Y 28.640, Z 27.200}
   LaserEnd_Ext()
   LIN {X 5.205, Y 29.640, Z 27.200}
   LaserStart_Ext()
   LIN {X -1.633, Y 29.640, Z 27.200}
   LaserEnd_Ext()
   LIN {X -1.779, Y 30.640, Z 27.200}
   LaserStart_Ext()
   LIN {X 4.953, Y 30.640, Z 27.200}
   LaserEnd_Ext()
   LIN {X 4.702, Y 31.640, Z 27.200}
   LaserStart_Ext()
   LIN {X -1.972, Y 31.640, Z 27.200}
   LaserEnd_Ext()
   LIN {X -2.166, Y 32.640, Z 27.200}
   LaserStart_Ext()
   LIN {X 4.438, Y 32.640, Z 27.200}
   LaserEnd_Ext()
   LIN {X 4.155, Y 33.640, Z 27.200}
   LaserStart_Ext()
   LIN {X -2.377, Y 33.640, Z 27.200}
   LaserEnd_Ext()
   LIN {X -2.605, Y 34.640, Z 27.200}
   LaserStart_Ext()
   LIN {X 3.871, Y 34.640, Z 27.200}
   LaserEnd_Ext()
   LIN {X 3.578, Y 35.640, Z 27.200}
   LaserStart_Ext()
   LIN {X -2.839, Y 35.640, Z 27.200}
   LaserEnd_Ext()
   LIN {X -3.096, Y 36.640, Z 27.200}
   LaserStart_Ext()
   LIN {X 3.270, Y 36.640, Z 27.200}
   LaserEnd_Ext()
   LIN {X 2.958, Y 37.640, Z 27.200}
   LaserStart_Ext()
   LIN {X -3.362, Y 37.640, Z 27.200}
   LaserEnd_Ext()
   LIN {X -3.540, Y 38.640, Z 27.200}
   LaserStart_Ext()
   LIN {X 2.632, Y 38.640, Z 27.200}
   LaserEnd_Ext()
   LIN {X 2.292, Y 39.640, Z 27.200}
   LaserStart_Ext()
   LIN {X -3.543, Y 39.640, Z 27.200}
   LaserEnd_Ext()
   LIN {X -3.160, Y 40.640, Z 27.200}
   LaserStart_Ext()
   LIN {X 1.790, Y 40.640, Z 27.200}
   LaserEnd_Ext()
   LIN {X 0.714, Y 41.640, Z 27.200}
   LaserStart_Ext()
   LIN {X -1.772, Y 41.640, Z 27.200}
   LaserEnd_Ext()
   LIN {X 1.702, Y -21.351, Z 28.050}
   LaserStart_Ext()
   LIN {X 1.701, Y -21.506, Z 28.050} C_DIS
   LIN {X 1.676, Y -23.527, Z 28.050} C_DIS
   LIN {X 0.710, Y -25.367, Z 28.050} C_DIS
   LIN {X 0.517, Y -25.741, Z 28.050} C_DIS
   LIN {X 0.192, Y -25.983, Z 28.050} C_DIS
   LIN {X -1.161, Y -26.974, Z 28.050} C_DIS
   LIN {X -2.893, Y -27.343, Z 28.050} C_DIS
   LIN {X -3.241, Y -27.416, Z 28.050} C_DIS
   LIN {X -3.720, Y -27.315, Z 28.050} C_DIS
   LIN {X -5.244, Y -26.998, Z 28.050} C_DIS
   LIN {X -6.220, Y -26.293, Z 28.050} C_DIS
   LIN {X -6.916, Y -25.786, Z 28.050} C_DIS
   LIN {X -7.416, Y -24.925, Z 28.050} C_DIS
   LIN {X -7.964, Y -23.986, Z 28.050} C_DIS
   LIN {X -8.069, Y -22.958, Z 28.050} C_DIS
   LIN {X -8.173, Y -21.909, Z 28.050} C_DIS
   LIN {X -7.535, Y -20.516, Z 28.050} C_DIS
   LIN {X -6.870, Y -19.041, Z 28.050} C_DIS
   LIN {X -5.771, Y -18.254, Z 28.050} C_DIS
   LIN {X -5.166, Y -17.824, Z 28.050} C_DIS
   LIN {X -4.676, Y -17.725, Z 28.050} C_DIS
   LIN {X -3.212, Y -17.414, Z 28.050} C_DIS
   LIN {X -1.175, Y -17.825, Z 28.050} C_DIS
   LIN {X 0.555, Y -19.081, Z 28.050} C_DIS
   LIN {X 1.602, Y -21.156, Z 28.050} C_DIS
   LIN {X 1.702, Y -21.351, Z 28.050}
   LaserEnd_Ext()
   LIN {X -2.461, Y 7.048, Z 28.050}
   LaserStart_Ext()
   LIN {X -2.585, Y 6.238, Z 28.050} C_DIS
   LIN {X -2.723, Y 5.401, Z 28.050} C_DIS
   LIN {X -3.264, Y 2.976, Z 28.050} C_DIS
   LIN {X -4.208, Y -1.343, Z 28.050} C_DIS
   LIN {X -5.154, Y -4.385, Z 28.050} C_DIS
   LIN {X -5.802, Y -6.462, Z 28.050} C_DIS
   LIN {X -6.346, Y -7.853, Z 28.050} C_DIS
   LIN {X -7.435, Y -10.682, Z 28.050} C_DIS
   LIN {X -8.827, Y -13.721, Z 28.050} C_DIS
   LIN {X -9.232, Y -14.595, Z 28.050} C_DIS
   LIN {X -9.670, Y -15.416, Z 28.050} C_DIS
   LIN {X -11.049, Y -18.031, Z 28.050} C_DIS
   LIN {X -11.607, Y -19.639, Z 28.050} C_DIS
   LIN {X -12.099, Y -21.022, Z 28.050} C_DIS
   LIN {X -11.959, Y -24.153, Z 28.050} C_DIS
   LIN {X -11.930, Y -24.729, Z 28.050} C_DIS
   LIN {X -11.791, Y -25.035, Z 28.050} C_DIS
   LIN {X -10.718, Y -27.438, Z 28.050} C_DIS
   LIN {X -8.741, Y -29.336, Z 28.050} C_DIS
   LIN {X -7.855, Y -30.161, Z 28.050} C_DIS
   LIN {X -5.281, Y -31.190, Z 28.050} C_DIS
   LIN {X -2.254, Y -31.367, Z 28.050} C_DIS
   LIN {X 0.891, Y -30.361, Z 28.050} C_DIS
   LIN {X 1.182, Y -30.256, Z 28.050} C_DIS
   LIN {X 1.341, Y -30.119, Z 28.050} C_DIS
   LIN {X 4.091, Y -27.647, Z 28.050} C_DIS
   LIN {X 4.790, Y -26.257, Z 28.050} C_DIS
   LIN {X 5.509, Y -24.693, Z 28.050} C_DIS
   LIN {X 6.226, Y -21.833, Z 28.050} C_DIS
   LIN {X 6.304, Y -21.528, Z 28.050} C_DIS
   LIN {X 6.339, Y -21.373, Z 28.050} C_DIS
   LIN {X 6.968, Y -18.538, Z 28.050} C_DIS
   LIN {X 7.372, Y -16.431, Z 28.050} C_DIS
   LIN {X 7.690, Y -14.716, Z 28.050} C_DIS
   LIN {X 8.194, Y -11.259, Z 28.050} C_DIS
   LIN {X 8.442, Y -9.596, Z 28.050} C_DIS
   LIN {X 8.529, Y -8.732, Z 28.050} C_DIS
   LIN {X 8.995, Y -3.877, Z 28.050} C_DIS
   LIN {X 9.111, Y -1.565, Z 28.050} C_DIS
   LIN {X 9.184, Y -0.153, Z 28.050} C_DIS
   LIN {X 9.238, Y 1.983, Z 28.050} C_DIS
   LIN {X 9.035, Y 10.455, Z 28.050} C_DIS
   LIN {X 8.942, Y 12.411, Z 28.050} C_DIS
   LIN {X 8.796, Y 13.811, Z 28.050} C_DIS
   LIN {X 7.763, Y 21.266, Z 28.050} C_DIS
   LIN {X 7.488, Y 23.501, Z 28.050} C_DIS
   LIN {X 7.351, Y 24.275, Z 28.050} C_DIS
   LIN {X 6.344, Y 29.035, Z 28.050} C_DIS
   LIN {X 6.281, Y 29.315, Z 28.050} C_DIS
   LIN {X 5.800, Y 31.225, Z 28.050} C_DIS
   LIN {X 5.544, Y 32.245, Z 28.050} C_DIS
   LIN {X 5.502, Y 32.400, Z 28.050} C_DIS
   LIN {X 4.783, Y 34.969, Z 28.050} C_DIS
   LIN {X 4.498, Y 35.919, Z 28.050} C_DIS
   LIN {X 3.999, Y 37.526, Z 28.050} C_DIS
   LIN {X 3.844, Y 38.006, Z 28.050} C_DIS
   LIN {X 3.520, Y 38.992, Z 28.050} C_DIS
   LIN {X 3.470, Y 39.138, Z 28.050} C_DIS
   LIN {X 3.034, Y 40.411, Z 28.050} C_DIS
   LIN {X 2.559, Y 41.241, Z 28.050} C_DIS
   LIN {X 2.302, Y 41.689, Z 28.050} C_DIS
   LIN {X 1.752, Y 42.104, Z 28.050} C_DIS
   LIN {X 0.914, Y 42.740, Z 28.050} C_DIS
   LIN {X 0.128, Y 42.910, Z 28.050} C_DIS
   LIN {X -0.793, Y 43.106, Z 28.050} C_DIS
   LIN {X -1.919, Y 42.712, Z 28.050} C_DIS
   LIN {X -3.168, Y 42.285, Z 28.050} C_DIS
   LIN {X -3.730, Y 41.647, Z 28.050} C_DIS
   LIN {X -4.249, Y 41.008, Z 28.050} C_DIS
   LIN {X -4.492, Y 40.211, Z 28.050} C_DIS
   LIN {X -4.693, Y 39.607, Z 28.050} C_DIS
   LIN {X -4.618, Y 38.735, Z 28.050} C_DIS
   LIN {X -4.555, Y 38.014, Z 28.050} C_DIS
   LIN {X -4.453, Y 37.646, Z 28.050} C_DIS
   LIN {X -4.225, Y 36.807, Z 28.050} C_DIS
   LIN {X -3.848, Y 35.357, Z 28.050} C_DIS
   LIN {X -3.823, Y 35.258, Z 28.050} C_DIS
   LIN {X -3.780, Y 35.070, Z 28.050} C_DIS
   LIN {X -3.290, Y 32.947, Z 28.050} C_DIS
   LIN {X -2.906, Y 30.983, Z 28.050} C_DIS
   LIN {X -2.792, Y 30.398, Z 28.050} C_DIS
   LIN {X -2.728, Y 29.961, Z 28.050} C_DIS
   LIN {X -2.495, Y 28.366, Z 28.050} C_DIS
   LIN {X -2.208, Y 26.475, Z 28.050} C_DIS
   LIN {X -1.877, Y 22.725, Z 28.050} C_DIS
   LIN {X -1.783, Y 21.626, Z 28.050} C_DIS
   LIN {X -1.805, Y 19.249, Z 28.050} C_DIS
   LIN {X -1.845, Y 12.642, Z 28.050} C_DIS
   LIN {X -2.067, Y 10.716, Z 28.050} C_DIS
   LIN {X -2.461, Y 7.048, Z 28.050}
   LaserEnd_Ext()
   LIN {X 7.602, Y -7.923, Z 28.050}
   LaserStart_Ext()
   LIN {X 7.602, Y 15.145, Z 28.050}
   LaserEnd_Ext()
   LIN {X 6.602, Y 22.517, Z 28.050}
   LaserStart_Ext()
   LIN {X 6.602, Y -15.100, Z 28.050}
   LaserEnd_Ext()
   LIN {X 5.602, Y -20.080, Z 28.050}
   LaserStart_Ext()
   LIN {X 5.602, Y 27.713, Z 28.050}
   LaserEnd_Ext()
   LIN {X 4.602, Y 31.891, Z 28.050}
   LaserStart_Ext()
   LIN {X 4.602, Y -24.198, Z 28.050}
   LaserEnd_Ext()
   LIN {X 3.602, Y -26.393, Z 28.050}
   LaserStart_Ext()
   LIN {X 3.602, Y 35.426, Z 28.050}
   LaserEnd_Ext()
   LIN {X 2.602, Y 38.583, Z 28.050}
   LaserStart_Ext()
   LIN {X 2.602, Y -20.917, Z 28.050}
   LaserEnd_Ext()
   LIN {X 2.602, Y -23.904, Z 28.050}
   LaserStart_Ext()
   LIN {X 2.602, Y -27.641, Z 28.050}
   LaserEnd_Ext()
   LIN {X 1.602, Y -28.540, Z 28.050}
   LaserStart_Ext()
   LIN {X 1.602, Y -25.820, Z 28.050}
   LaserEnd_Ext()
   LIN {X 1.602, Y -18.936, Z 28.050}
   LaserStart_Ext()
   LIN {X 1.602, Y 40.900, Z 28.050}
   LaserEnd_Ext()
   LIN {X 0.602, Y 41.722, Z 28.050}
   LaserStart_Ext()
   LIN {X 0.602, Y -17.877, Z 28.050}
   LaserEnd_Ext()
   LIN {X 0.602, Y -26.922, Z 28.050}
   LaserStart_Ext()
   LIN {X 0.602, Y -29.402, Z 28.050}
   LaserEnd_Ext()
   LIN {X -0.398, Y -29.723, Z 28.050}
   LaserStart_Ext()
   LIN {X -0.398, Y -27.655, Z 28.050}
   LaserEnd_Ext()
   LIN {X -0.398, Y -17.146, Z 28.050}
   LaserStart_Ext()
   LIN {X -0.398, Y 41.999, Z 28.050}
   LaserEnd_Ext()
   LIN {X -1.398, Y 41.834, Z 28.050}
   LaserStart_Ext()
   LIN {X -1.398, Y 27.805, Z 28.050}
   LaserEnd_Ext()
   LIN {X -1.398, Y 7.579, Z 28.050}
   LaserStart_Ext()
   LIN {X -1.398, Y -16.760, Z 28.050}
   LaserEnd_Ext()
   LIN {X -1.398, Y -28.047, Z 28.050}
   LaserStart_Ext()
   LIN {X -1.398, Y -30.043, Z 28.050}
   LaserEnd_Ext()
   LIN {X -2.398, Y -30.357, Z 28.050}
   LaserStart_Ext()
   LIN {X -2.398, Y -28.260, Z 28.050}
   LaserEnd_Ext()
   LIN {X -2.398, Y -16.558, Z 28.050}
   LaserStart_Ext()
   LIN {X -2.398, Y 2.256, Z 28.050}
   LaserEnd_Ext()
   LIN {X -2.398, Y 33.531, Z 28.050}
   LaserStart_Ext()
   LIN {X -2.398, Y 41.492, Z 28.050}
   LaserEnd_Ext()
   LIN {X -3.398, Y 40.370, Z 28.050}
   LaserStart_Ext()
   LIN {X -3.398, Y 37.577, Z 28.050}
   LaserEnd_Ext()
   LIN {X -3.398, Y -2.107, Z 28.050}
   LaserStart_Ext()
   LIN {X -3.398, Y -16.432, Z 28.050}
   LaserEnd_Ext()
   LIN {X -3.398, Y -28.402, Z 28.050}
   LaserStart_Ext()
   LIN {X -3.398, Y -30.303, Z 28.050}
   LaserEnd_Ext()
   LIN {X -4.398, Y -30.248, Z 28.050}
   LaserStart_Ext()
   LIN {X -4.398, Y -28.195, Z 28.050}
   LaserEnd_Ext()
   LIN {X -4.398, Y -16.643, Z 28.050}
   LaserStart_Ext()
   LIN {X -4.398, Y -5.320, Z 28.050}
   LaserEnd_Ext()
   LIN {X -5.398, Y -8.176, Z 28.050}
   LaserStart_Ext()
   LIN {X -5.398, Y -16.853, Z 28.050}
   LaserEnd_Ext()
   LIN {X -5.398, Y -27.987, Z 28.050}
   LaserStart_Ext()
   LIN {X -5.398, Y -30.066, Z 28.050}
   LaserEnd_Ext()
   LIN {X -6.398, Y -29.666, Z 28.050}
   LaserStart_Ext()
   LIN {X -6.398, Y -27.398, Z 28.050}
   LaserEnd_Ext()
   LIN {X -6.398, Y -17.473, Z 28.050}
   LaserStart_Ext()
   LIN {X -6.398, Y -10.772, Z 28.050}
   LaserEnd_Ext()
   LIN {X -7.398, Y -13.003, Z 28.050}
   LaserStart_Ext()
   LIN {X -7.398, Y -18.189, Z 28.050}
   LaserEnd_Ext()
   LIN {X -7.398, Y -26.672, Z 28.050}
   LaserStart_Ext()
   LIN {X -7.398, Y -29.220, Z 28.050}
   LaserEnd_Ext()
   LIN {X -8.398, Y -28.279, Z 28.050}
   LaserStart_Ext()
   LIN {X -8.398, Y -25.225, Z 28.050}
   LaserEnd_Ext()
   LIN {X -8.398, Y -19.998, Z 28.050}
   LaserStart_Ext()
   LIN {X -8.398, Y -15.157, Z 28.050}
   LaserEnd_Ext()
   LIN {X -9.398, Y -17.044, Z 28.050}
   LaserStart_Ext()
   LIN {X -9.398, Y -27.319, Z 28.050}
   LaserEnd_Ext()
   LIN {X -10.398, Y -25.703, Z 28.050}
   LaserStart_Ext()
   LIN {X -10.398, Y -19.206, Z 28.050}
   LaserEnd_Ext()
   LIN {X -8.053, Y -22.307, Z 28.900}
   LaserStart_Ext()
   LIN {X -8.099, Y -21.874, Z 28.900} C_DIS
   LIN {X -7.829, Y -21.264, Z 28.900} C_DIS
   LIN {X -6.815, Y -19.017, Z 28.900} C_DIS
   LIN {X -5.693, Y -18.213, Z 28.900} C_DIS
   LIN {X -5.120, Y -17.790, Z 28.900} C_DIS
   LIN {X -4.135, Y -17.568, Z 28.900} C_DIS
   LIN {X -3.191, Y -17.367, Z 28.900} C_DIS
   LIN {X -2.458, Y -17.515, Z 28.900} C_DIS
   LIN {X -1.095, Y -17.776, Z 28.900} C_DIS
   LIN {X 0.263, Y -18.763, Z 28.900} C_DIS
   LIN {X 0.623, Y -19.025, Z 28.900} C_DIS
   LIN {X 0.844, Y -19.464, Z 28.900} C_DIS
   LIN {X 1.775, Y -21.293, Z 28.900} C_DIS
   LIN {X 1.763, Y -22.736, Z 28.900} C_DIS
   LIN {X 1.754, Y -23.469, Z 28.900} C_DIS
   LIN {X 1.404, Y -24.136, Z 28.900} C_DIS
   LIN {X 0.610, Y -25.674, Z 28.900} C_DIS
   LIN {X -0.731, Y -26.671, Z 28.900} C_DIS
   LIN {X -1.075, Y -26.923, Z 28.900} C_DIS
   LIN {X -1.739, Y -27.064, Z 28.900} C_DIS
   LIN {X -3.146, Y -27.369, Z 28.900} C_DIS
   LIN {X -4.084, Y -27.179, Z 28.900} C_DIS
   LIN {X -5.158, Y -26.955, Z 28.900} C_DIS
   LIN {X -6.313, Y -26.121, Z 28.900} C_DIS
   LIN {X -6.833, Y -25.747, Z 28.900} C_DIS
   LIN {X -7.092, Y -25.308, Z 28.900} C_DIS
   LIN {X -7.885, Y -23.950, Z 28.900} C_DIS
   LIN {X -8.053, Y -22.307, Z 28.900}
   LaserEnd_Ext()
   LIN {X -9.180, Y -14.573, Z 28.900}
   LaserStart_Ext()
   LIN {X -9.444, Y -15.083, Z 28.900} C_DIS
   LIN {X -10.983, Y -18.002, Z 28.900} C_DIS
   LIN {X -11.854, Y -20.509, Z 28.900} C_DIS
   LIN {X -12.027, Y -20.996, Z 28.900} C_DIS
   LIN {X -11.978, Y -22.098, Z 28.900} C_DIS
   LIN {X -11.849, Y -24.702, Z 28.900} C_DIS
   LIN {X -11.220, Y -26.089, Z 28.900} C_DIS
   LIN {X -10.631, Y -27.409, Z 28.900} C_DIS
   LIN {X -9.545, Y -28.451, Z 28.900} C_DIS
   LIN {X -7.723, Y -30.146, Z 28.900} C_DIS
   LIN {X -5.820, Y -30.907, Z 28.900} C_DIS
   LIN {X -5.046, Y -31.181, Z 28.900} C_DIS
   LIN {X -4.173, Y -31.218, Z 28.900} C_DIS
   LIN {X -2.226, Y -31.325, Z 28.900} C_DIS
   LIN {X 0.273, Y -30.526, Z 28.900} C_DIS
   LIN {X 1.305, Y -30.182, Z 28.900} C_DIS
   LIN {X 3.966, Y -27.727, Z 28.900} C_DIS
   LIN {X 4.295, Y -27.431, Z 28.900} C_DIS
   LIN {X 4.353, Y -27.317, Z 28.900} C_DIS
   LIN {X 5.590, Y -24.625, Z 28.900} C_DIS
   LIN {X 6.134, Y -22.460, Z 28.900} C_DIS
   LIN {X 6.378, Y -21.459, Z 28.900} C_DIS
   LIN {X 6.834, Y -19.370, Z 28.900} C_DIS
   LIN {X 7.035, Y -18.467, Z 28.900} C_DIS
   LIN {X 7.143, Y -17.899, Z 28.900} C_DIS
   LIN {X 7.748, Y -14.644, Z 28.900} C_DIS
   LIN {X 8.339, Y -10.590, Z 28.900} C_DIS
   LIN {X 8.474, Y -9.638, Z 28.900} C_DIS
   LIN {X 8.656, Y -7.693, Z 28.900} C_DIS
   LIN {X 9.019, Y -3.918, Z 28.900} C_DIS
   LIN {X 9.075, Y -2.798, Z 28.900} C_DIS
   LIN {X 9.179, Y -0.787, Z 28.900} C_DIS
   LIN {X 9.256, Y 2.254, Z 28.900} C_DIS
   LIN {X 9.078, Y 9.654, Z 28.900} C_DIS
   LIN {X 8.953, Y 12.295, Z 28.900} C_DIS
   LIN {X 8.757, Y 14.185, Z 28.900} C_DIS
   LIN {X 7.460, Y 23.542, Z 28.900} C_DIS
   LIN {X 7.422, Y 23.797, Z 28.900} C_DIS
   LIN {X 7.400, Y 23.898, Z 28.900} C_DIS
   LIN {X 7.362, Y 24.053, Z 28.900} C_DIS
   LIN {X 7.328, Y 24.222, Z 28.900} C_DIS
   LIN {X 6.209, Y 29.479, Z 28.900} C_DIS
   LIN {X 5.656, Y 31.684, Z 28.900} C_DIS
   LIN {X 5.316, Y 32.942, Z 28.900} C_DIS
   LIN {X 4.894, Y 34.447, Z 28.900} C_DIS
   LIN {X 4.347, Y 36.275, Z 28.900} C_DIS
   LIN {X 4.216, Y 36.698, Z 28.900} C_DIS
   LIN {X 3.681, Y 38.358, Z 28.900} C_DIS
   LIN {X 3.517, Y 38.859, Z 28.900} C_DIS
   LIN {X 3.094, Y 40.087, Z 28.900} C_DIS
   LIN {X 2.961, Y 40.473, Z 28.900} C_DIS
   LIN {X 2.772, Y 40.800, Z 28.900} C_DIS
   LIN {X 2.226, Y 41.748, Z 28.900} C_DIS
   LIN {X 1.300, Y 42.448, Z 28.900} C_DIS
   LIN {X 0.836, Y 42.797, Z 28.900} C_DIS
   LIN {X -0.061, Y 42.986, Z 28.900} C_DIS
   LIN {X -0.872, Y 43.158, Z 28.900} C_DIS
   LIN {X -2.368, Y 42.635, Z 28.900} C_DIS
   LIN {X -3.281, Y 42.304, Z 28.900} C_DIS
   LIN {X -3.670, Y 41.802, Z 28.900} C_DIS
   LIN {X -4.401, Y 40.900, Z 28.900} C_DIS
   LIN {X -4.575, Y 40.333, Z 28.900} C_DIS
   LIN {X -4.769, Y 39.587, Z 28.900} C_DIS
   LIN {X -4.693, Y 38.869, Z 28.900} C_DIS
   LIN {X -4.622, Y 38.058, Z 28.900} C_DIS
   LIN {X -4.361, Y 37.110, Z 28.900} C_DIS
   LIN {X -4.289, Y 36.852, Z 28.900} C_DIS
   LIN {X -4.227, Y 36.618, Z 28.900} C_DIS
   LIN {X -3.883, Y 35.303, Z 28.900} C_DIS
   LIN {X -3.369, Y 33.096, Z 28.900} C_DIS
   LIN {X -3.345, Y 32.994, Z 28.900} C_DIS
   LIN {X -2.817, Y 30.310, Z 28.900} C_DIS
   LIN {X -2.657, Y 29.219, Z 28.900} C_DIS
   LIN {X -2.244, Y 26.497, Z 28.900} C_DIS
   LIN {X -1.855, Y 22.090, Z 28.900} C_DIS
   LIN {X -1.803, Y 21.536, Z 28.900} C_DIS
   LIN {X -1.802, Y 21.302, Z 28.900} C_DIS
   LIN {X -1.855, Y 12.638, Z 28.900} C_DIS
   LIN {X -2.185, Y 9.776, Z 28.900} C_DIS
   LIN {X -2.517, Y 6.679, Z 28.900} C_DIS
   LIN {X -2.668, Y 5.693, Z 28.900} C_DIS
   LIN {X -2.695, Y 5.562, Z 28.900} C_DIS
   LIN {X -4.243, Y -1.526, Z 28.900} C_DIS
   LIN {X -5.772, Y -6.441, Z 28.900} C_DIS
   LIN {X -7.408, Y -10.696, Z 28.900} C_DIS
   LIN {X -8.936, Y -14.031, Z 28.900} C_DIS
   LIN {X -9.180, Y -14.573, Z 28.900}
   LaserEnd_Ext()
   LIN {X -2.504, Y 41.522, Z 28.900}
   LaserStart_Ext()
   LIN {X 0.867, Y 41.522, Z 28.900}
   LaserEnd_Ext()
   LIN {X 1.778, Y 40.522, Z 28.900}
   LaserStart_Ext()
   LIN {X -3.421, Y 40.522, Z 28.900}
   LaserEnd_Ext()
   LIN {X -3.753, Y 39.522, Z 28.900}
   LaserStart_Ext()
   LIN {X 2.231, Y 39.522, Z 28.900}
   LaserEnd_Ext()
   LIN {X 2.575, Y 38.522, Z 28.900}
   LaserStart_Ext()
   LIN {X -3.659, Y 38.522, Z 28.900}
   LaserEnd_Ext()
   LIN {X -3.437, Y 37.522, Z 28.900}
   LaserStart_Ext()
   LIN {X 2.900, Y 37.522, Z 28.900}
   LaserEnd_Ext()
   LIN {X 3.222, Y 36.522, Z 28.900}
   LaserStart_Ext()
   LIN {X -3.168, Y 36.522, Z 28.900}
   LaserEnd_Ext()
   LIN {X -2.907, Y 35.522, Z 28.900}
   LaserStart_Ext()
   LIN {X 3.529, Y 35.522, Z 28.900}
   LaserEnd_Ext()
   LIN {X 3.828, Y 34.522, Z 28.900}
   LaserStart_Ext()
   LIN {X -2.674, Y 34.522, Z 28.900}
   LaserEnd_Ext()
   LIN {X -2.441, Y 33.522, Z 28.900}
   LaserStart_Ext()
   LIN {X 4.115, Y 33.522, Z 28.900}
   LaserEnd_Ext()
   LIN {X 4.394, Y 32.522, Z 28.900}
   LaserStart_Ext()
   LIN {X -2.233, Y 32.522, Z 28.900}
   LaserEnd_Ext()
   LIN {X -2.036, Y 31.522, Z 28.900}
   LaserStart_Ext()
   LIN {X 4.664, Y 31.522, Z 28.900}
   LaserEnd_Ext()
   LIN {X 4.917, Y 30.522, Z 28.900}
   LaserStart_Ext()
   LIN {X -1.840, Y 30.522, Z 28.900}
   LaserEnd_Ext()
   LIN {X -1.691, Y 29.522, Z 28.900}
   LaserStart_Ext()
   LIN {X 5.167, Y 29.522, Z 28.900}
   LaserEnd_Ext()
   LIN {X 5.390, Y 28.522, Z 28.900}
   LaserStart_Ext()
   LIN {X -1.540, Y 28.522, Z 28.900}
   LaserEnd_Ext()
   LIN {X -1.388, Y 27.522, Z 28.900}
   LaserStart_Ext()
   LIN {X 5.603, Y 27.522, Z 28.900}
   LaserEnd_Ext()
   LIN {X 5.816, Y 26.522, Z 28.900}
   LaserStart_Ext()
   LIN {X -1.243, Y 26.522, Z 28.900}
   LaserEnd_Ext()
   LIN {X -1.154, Y 25.522, Z 28.900}
   LaserStart_Ext()
   LIN {X 6.029, Y 25.522, Z 28.900}
   LaserEnd_Ext()
   LIN {X 6.242, Y 24.522, Z 28.900}
   LaserStart_Ext()
   LIN {X -1.066, Y 24.522, Z 28.900}
   LaserEnd_Ext()
   LIN {X -0.978, Y 23.522, Z 28.900}
   LaserStart_Ext()
   LIN {X 6.452, Y 23.522, Z 28.900}
   LaserEnd_Ext()
   LIN {X 6.592, Y 22.522, Z 28.900}
   LaserStart_Ext()
   LIN {X -0.889, Y 22.522, Z 28.900}
   LaserEnd_Ext()
   LIN {X -0.803, Y 21.522, Z 28.900}
   LaserStart_Ext()
   LIN {X 6.731, Y 21.522, Z 28.900}
   LaserEnd_Ext()
   LIN {X 6.869, Y 20.522, Z 28.900}
   LaserStart_Ext()
   LIN {X -0.807, Y 20.522, Z 28.900}
   LaserEnd_Ext()
   LIN {X -0.813, Y 19.522, Z 28.900}
   LaserStart_Ext()
   LIN {X 7.008, Y 19.522, Z 28.900}
   LaserEnd_Ext()
   LIN {X 7.146, Y 18.522, Z 28.900}
   LaserStart_Ext()
   LIN {X -0.819, Y 18.522, Z 28.900}
   LaserEnd_Ext()
   LIN {X -0.825, Y 17.522, Z 28.900}
   LaserStart_Ext()
   LIN {X 7.285, Y 17.522, Z 28.900}
   LaserEnd_Ext()
   LIN {X 7.423, Y 16.522, Z 28.900}
   LaserStart_Ext()
   LIN {X -0.831, Y 16.522, Z 28.900}
   LaserEnd_Ext()
   LIN {X -0.837, Y 15.522, Z 28.900}
   LaserStart_Ext()
   LIN {X 7.562, Y 15.522, Z 28.900}
   LaserEnd_Ext()
   LIN {X 7.700, Y 14.522, Z 28.900}
   LaserStart_Ext()
   LIN {X -0.843, Y 14.522, Z 28.900}
   LaserEnd_Ext()
   LIN {X -0.850, Y 13.522, Z 28.900}
   LaserStart_Ext()
   LIN {X 7.820, Y 13.522, Z 28.900}
   LaserEnd_Ext()
   LIN {X 7.924, Y 12.522, Z 28.900}
   LaserStart_Ext()
   LIN {X -0.862, Y 12.522, Z 28.900}
   LaserEnd_Ext()
   LIN {X -0.977, Y 11.522, Z 28.900}
   LaserStart_Ext()
   LIN {X 7.989, Y 11.522, Z 28.900}
   LaserEnd_Ext()
   LIN {X 8.036, Y 10.522, Z 28.900}
   LaserStart_Ext()
   LIN {X -1.092, Y 10.522, Z 28.900}
   LaserEnd_Ext()
   LIN {X -1.206, Y 9.522, Z 28.900}
   LaserStart_Ext()
   LIN {X 8.081, Y 9.522, Z 28.900}
   LaserEnd_Ext()
   LIN {X 8.105, Y 8.522, Z 28.900}
   LaserStart_Ext()
   LIN {X -1.313, Y 8.522, Z 28.900}
   LaserEnd_Ext()
   LIN {X -1.421, Y 7.522, Z 28.900}
   LaserStart_Ext()
   LIN {X 8.129, Y 7.522, Z 28.900}
   LaserEnd_Ext()
   LIN {X 8.153, Y 6.522, Z 28.900}
   LaserStart_Ext()
   LIN {X -1.529, Y 6.522, Z 28.900}
   LaserEnd_Ext()
   LIN {X -1.683, Y 5.522, Z 28.900}
   LaserStart_Ext()
   LIN {X 8.177, Y 5.522, Z 28.900}
   LaserEnd_Ext()
   LIN {X 8.201, Y 4.522, Z 28.900}
   LaserStart_Ext()
   LIN {X -1.899, Y 4.522, Z 28.900}
   LaserEnd_Ext()
   LIN {X -2.117, Y 3.522, Z 28.900}
   LaserStart_Ext()
   LIN {X 8.225, Y 3.522, Z 28.900}
   LaserEnd_Ext()
   LIN {X 8.250, Y 2.522, Z 28.900}
   LaserStart_Ext()
   LIN {X -2.336, Y 2.522, Z 28.900}
   LaserEnd_Ext()
   LIN {X -2.554, Y 1.522, Z 28.900}
   LaserStart_Ext()
   LIN {X 8.237, Y 1.522, Z 28.900}
   LaserEnd_Ext()
   LIN {X 8.212, Y 0.522, Z 28.900}
   LaserStart_Ext()
   LIN {X -2.772, Y 0.522, Z 28.900}
   LaserEnd_Ext()
   LIN {X -2.991, Y -0.478, Z 28.900}
   LaserStart_Ext()
   LIN {X 8.186, Y -0.478, Z 28.900}
   LaserEnd_Ext()
   LIN {X 8.142, Y -1.478, Z 28.900}
   LaserStart_Ext()
   LIN {X -3.209, Y -1.478, Z 28.900}
   LaserEnd_Ext()
   LIN {X -3.492, Y -2.478, Z 28.900}
   LaserStart_Ext()
   LIN {X 8.090, Y -2.478, Z 28.900}
   LaserEnd_Ext()
   LIN {X 8.040, Y -3.478, Z 28.900}
   LaserStart_Ext()
   LIN {X -3.803, Y -3.478, Z 28.900}
   LaserEnd_Ext()
   LIN {X -4.114, Y -4.478, Z 28.900}
   LaserStart_Ext()
   LIN {X 7.960, Y -4.478, Z 28.900}
   LaserEnd_Ext()
   LIN {X 7.864, Y -5.478, Z 28.900}
   LaserStart_Ext()
   LIN {X -4.426, Y -5.478, Z 28.900}
   LaserEnd_Ext()
   LIN {X -4.737, Y -6.478, Z 28.900}
   LaserStart_Ext()
   LIN {X 7.768, Y -6.478, Z 28.900}
   LaserEnd_Ext()
   LIN {X 7.672, Y -7.478, Z 28.900}
   LaserStart_Ext()
   LIN {X -5.098, Y -7.478, Z 28.900}
   LaserEnd_Ext()
   LIN {X -5.483, Y -8.478, Z 28.900}
   LaserStart_Ext()
   LIN {X 7.578, Y -8.478, Z 28.900}
   LaserEnd_Ext()
   LIN {X 7.484, Y -9.478, Z 28.900}
   LaserStart_Ext()
   LIN {X -5.868, Y -9.478, Z 28.900}
   LaserEnd_Ext()
   LIN {X -6.253, Y -10.478, Z 28.900}
   LaserStart_Ext()
   LIN {X 7.345, Y -10.478, Z 28.900}
   LaserEnd_Ext()
   LIN {X 7.199, Y -11.478, Z 28.900}
   LaserStart_Ext()
   LIN {X -6.667, Y -11.478, Z 28.900}
   LaserEnd_Ext()
   LIN {X -7.125, Y -12.478, Z 28.900}
   LaserStart_Ext()
   LIN {X 7.053, Y -12.478, Z 28.900}
   LaserEnd_Ext()
   LIN {X 6.907, Y -13.478, Z 28.900}
   LaserStart_Ext()
   LIN {X -7.583, Y -13.478, Z 28.900}
   LaserEnd_Ext()
   LIN {X -8.040, Y -14.478, Z 28.900}
   LaserStart_Ext()
   LIN {X 6.761, Y -14.478, Z 28.900}
   LaserEnd_Ext()
   LIN {X 6.576, Y -15.478, Z 28.900}
   LaserStart_Ext()
   LIN {X -8.523, Y -15.478, Z 28.900}
   LaserEnd_Ext()
   LIN {X -9.050, Y -16.478, Z 28.900}
   LaserStart_Ext()
   LIN {X -3.818, Y -16.478, Z 28.900}
   LaserEnd_Ext()
   LIN {X -2.540, Y -16.478, Z 28.900}
   LaserStart_Ext()
   LIN {X 6.390, Y -16.478, Z 28.900}
   LaserEnd_Ext()
   LIN {X 6.204, Y -17.478, Z 28.900}
   LaserStart_Ext()
   LIN {X 0.197, Y -17.478, Z 28.900}
   LaserEnd_Ext()
   LIN {X -6.385, Y -17.478, Z 28.900}
   LaserStart_Ext()
   LIN {X -9.577, Y -17.478, Z 28.900}
   LaserEnd_Ext()
   LIN {X -10.090, Y -18.478, Z 28.900}
   LaserStart_Ext()
   LIN {X -7.656, Y -18.478, Z 28.900}
   LaserEnd_Ext()
   LIN {X 1.459, Y -18.478, Z 28.900}
   LaserStart_Ext()
   LIN {X 6.008, Y -18.478, Z 28.900}
   LaserEnd_Ext()
   LIN {X 5.787, Y -19.478, Z 28.900}
   LaserStart_Ext()
   LIN {X 1.973, Y -19.478, Z 28.900}
   LaserEnd_Ext()
   LIN {X -8.120, Y -19.478, Z 28.900}
   LaserStart_Ext()
   LIN {X -10.437, Y -19.478, Z 28.900}
   LaserEnd_Ext()
   LIN {X -10.785, Y -20.478, Z 28.900}
   LaserStart_Ext()
   LIN {X -8.571, Y -20.478, Z 28.900}
   LaserEnd_Ext()
   LIN {X 2.482, Y -20.478, Z 28.900}
   LaserStart_Ext()
   LIN {X 5.569, Y -20.478, Z 28.900}
   LaserEnd_Ext()
   LIN {X 5.344, Y -21.478, Z 28.900}
   LaserStart_Ext()
   LIN {X 2.773, Y -21.478, Z 28.900}
   LaserEnd_Ext()
   LIN {X -9.017, Y -21.478, Z 28.900}
   LaserStart_Ext()
   LIN {X -11.004, Y -21.478, Z 28.900}
   LaserEnd_Ext()
   LIN {X -10.958, Y -22.478, Z 28.900}
   LaserStart_Ext()
   LIN {X -9.041, Y -22.478, Z 28.900}
   LaserEnd_Ext()
   LIN {X 2.765, Y -22.478, Z 28.900}
   LaserStart_Ext()
   LIN {X 5.098, Y -22.478, Z 28.900}
   LaserEnd_Ext()
   LIN {X 4.847, Y -23.478, Z 28.900}
   LaserStart_Ext()
   LIN {X 2.754, Y -23.478, Z 28.900}
   LaserEnd_Ext()
   LIN {X -8.938, Y -23.478, Z 28.900}
   LaserStart_Ext()
   LIN {X -10.908, Y -23.478, Z 28.900}
   LaserEnd_Ext()
   LIN {X -10.852, Y -24.478, Z 28.900}
   LaserStart_Ext()
   LIN {X -8.734, Y -24.478, Z 28.900}
   LaserEnd_Ext()
   LIN {X 2.353, Y -24.478, Z 28.900}
   LaserStart_Ext()
   LIN {X 4.557, Y -24.478, Z 28.900}
   LaserEnd_Ext()
   LIN {X 4.097, Y -25.478, Z 28.900}
   LaserStart_Ext()
   LIN {X 1.836, Y -25.478, Z 28.900}
   LaserEnd_Ext()
   LIN {X -8.150, Y -25.478, Z 28.900}
   LaserStart_Ext()
   LIN {X -10.399, Y -25.478, Z 28.900}
   LaserEnd_Ext()
   LIN {X -9.951, Y -26.478, Z 28.900}
   LaserStart_Ext()
   LIN {X -7.514, Y -26.478, Z 28.900}
   LaserEnd_Ext()
   LIN {X 1.205, Y -26.478, Z 28.900}
   LaserStart_Ext()
   LIN {X 3.638, Y -26.478, Z 28.900}
   LaserEnd_Ext()
   LIN {X 2.761, Y -27.478, Z 28.900}
   LaserStart_Ext()
   LIN {X -0.142, Y -27.478, Z 28.900}
   LaserEnd_Ext()
   LIN {X -6.142, Y -27.478, Z 28.900}
   LaserStart_Ext()
   LIN {X -9.115, Y -27.478, Z 28.900}
   LaserEnd_Ext()
   LIN {X -8.048, Y -28.478, Z 28.900}
   LaserStart_Ext()
   LIN {X 1.677, Y -28.478, Z 28.900}
   LaserEnd_Ext()
   LIN {X 0.254, Y -29.478, Z 28.900}
   LaserStart_Ext()
   LIN {X -6.700, Y -29.478, Z 28.900}
   LaserEnd_Ext()
   LIN {X -0.980, Y -26.866, Z 29.750}
   LaserStart_Ext()
   LIN {X -1.781, Y -27.047, Z 29.750} C_DIS
   LIN {X -3.047, Y -27.322, Z 29.750} C_DIS
   LIN {X -4.798, Y -26.967, Z 29.750} C_DIS
   LIN {X -5.072, Y -26.913, Z 29.750} C_DIS
   LIN {X -5.239, Y -26.794, Z 29.750} C_DIS
   LIN {X -6.750, Y -25.709, Z 29.750} C_DIS
   LIN {X -7.696, Y -24.101, Z 29.750} C_DIS
   LIN {X -7.806, Y -23.914, Z 29.750} C_DIS
   LIN {X -7.829, Y -23.687, Z 29.750} C_DIS
   LIN {X -8.025, Y -21.838, Z 29.750} C_DIS
   LIN {X -6.869, Y -19.233, Z 29.750} C_DIS
   LIN {X -6.761, Y -18.992, Z 29.750} C_DIS
   LIN {X -6.640, Y -18.906, Z 29.750} C_DIS
   LIN {X -5.093, Y -17.765, Z 29.750} C_DIS
   LIN {X -3.662, Y -17.442, Z 29.750} C_DIS
   LIN {X -3.148, Y -17.320, Z 29.750} C_DIS
   LIN {X -2.416, Y -17.459, Z 29.750} C_DIS
   LIN {X -1.031, Y -17.724, Z 29.750} C_DIS
   LIN {X -0.119, Y -18.386, Z 29.750} C_DIS
   LIN {X 0.690, Y -18.969, Z 29.750} C_DIS
   LIN {X 1.230, Y -20.020, Z 29.750} C_DIS
   LIN {X 1.848, Y -21.234, Z 29.750} C_DIS
   LIN {X 1.836, Y -22.674, Z 29.750} C_DIS
   LIN {X 1.832, Y -23.410, Z 29.750} C_DIS
   LIN {X 1.288, Y -24.473, Z 29.750} C_DIS
   LIN {X 0.703, Y -25.608, Z 29.750} C_DIS
   LIN {X 0.010, Y -26.122, Z 29.750} C_DIS
   LIN {X -0.980, Y -26.866, Z 29.750}
   LaserEnd_Ext()
   LIN {X 9.032, Y -4.078, Z 29.750}
   LaserStart_Ext()
   LIN {X 9.043, Y -3.959, Z 29.750} C_DIS
   LIN {X 9.174, Y -1.422, Z 29.750} C_DIS
   LIN {X 9.274, Y 2.524, Z 29.750} C_DIS
   LIN {X 9.122, Y 8.852, Z 29.750} C_DIS
   LIN {X 8.965, Y 12.178, Z 29.750} C_DIS
   LIN {X 8.717, Y 14.559, Z 29.750} C_DIS
   LIN {X 7.732, Y 21.664, Z 29.750} C_DIS
   LIN {X 7.429, Y 23.666, Z 29.750} C_DIS
   LIN {X 7.257, Y 24.458, Z 29.750} C_DIS
   LIN {X 6.966, Y 25.673, Z 29.750} C_DIS
   LIN {X 6.694, Y 26.993, Z 29.750} C_DIS
   LIN {X 6.074, Y 29.903, Z 29.750} C_DIS
   LIN {X 5.769, Y 31.123, Z 29.750} C_DIS
   LIN {X 5.130, Y 33.484, Z 29.750} C_DIS
   LIN {X 5.006, Y 33.926, Z 29.750} C_DIS
   LIN {X 4.755, Y 34.766, Z 29.750} C_DIS
   LIN {X 4.339, Y 36.168, Z 29.750} C_DIS
   LIN {X 4.193, Y 36.630, Z 29.750} C_DIS
   LIN {X 3.553, Y 38.604, Z 29.750} C_DIS
   LIN {X 3.518, Y 38.710, Z 29.750} C_DIS
   LIN {X 2.888, Y 40.534, Z 29.750} C_DIS
   LIN {X 2.278, Y 41.589, Z 29.750} C_DIS
   LIN {X 2.150, Y 41.807, Z 29.750} C_DIS
   LIN {X 1.837, Y 42.042, Z 29.750} C_DIS
   LIN {X 0.758, Y 42.853, Z 29.750} C_DIS
   LIN {X -0.112, Y 43.036, Z 29.750} C_DIS
   LIN {X -0.951, Y 43.210, Z 29.750} C_DIS
   LIN {X -2.446, Y 42.637, Z 29.750} C_DIS
   LIN {X -3.451, Y 42.273, Z 29.750} C_DIS
   LIN {X -3.927, Y 41.659, Z 29.750} C_DIS
   LIN {X -4.533, Y 40.820, Z 29.750} C_DIS
   LIN {X -4.726, Y 39.992, Z 29.750} C_DIS
   LIN {X -4.850, Y 39.516, Z 29.750} C_DIS
   LIN {X -4.781, Y 38.864, Z 29.750} C_DIS
   LIN {X -4.689, Y 38.101, Z 29.750} C_DIS
   LIN {X -4.554, Y 37.621, Z 29.750} C_DIS
   LIN {X -4.353, Y 36.896, Z 29.750} C_DIS
   LIN {X -4.009, Y 35.595, Z 29.750} C_DIS
   LIN {X -3.944, Y 35.349, Z 29.750} C_DIS
   LIN {X -3.878, Y 35.072, Z 29.750} C_DIS
   LIN {X -3.400, Y 33.040, Z 29.750} C_DIS
   LIN {X -2.911, Y 30.575, Z 29.750} C_DIS
   LIN {X -2.842, Y 30.221, Z 29.750} C_DIS
   LIN {X -2.820, Y 30.072, Z 29.750} C_DIS
   LIN {X -2.281, Y 26.519, Z 29.750} C_DIS
   LIN {X -2.057, Y 23.988, Z 29.750} C_DIS
   LIN {X -1.823, Y 21.463, Z 29.750} C_DIS
   LIN {X -1.817, Y 20.400, Z 29.750} C_DIS
   LIN {X -1.865, Y 12.635, Z 29.750} C_DIS
   LIN {X -2.302, Y 8.836, Z 29.750} C_DIS
   LIN {X -2.573, Y 6.310, Z 29.750} C_DIS
   LIN {X -2.698, Y 5.493, Z 29.750} C_DIS
   LIN {X -3.248, Y 3.009, Z 29.750} C_DIS
   LIN {X -4.278, Y -1.708, Z 29.750} C_DIS
   LIN {X -5.265, Y -4.880, Z 29.750} C_DIS
   LIN {X -5.762, Y -6.485, Z 29.750} C_DIS
   LIN {X -6.379, Y -8.107, Z 29.750} C_DIS
   LIN {X -7.382, Y -10.710, Z 29.750} C_DIS
   LIN {X -8.331, Y -12.782, Z 29.750} C_DIS
   LIN {X -9.127, Y -14.551, Z 29.750} C_DIS
   LIN {X -9.991, Y -16.215, Z 29.750} C_DIS
   LIN {X -10.918, Y -17.974, Z 29.750} C_DIS
   LIN {X -11.717, Y -20.275, Z 29.750} C_DIS
   LIN {X -11.955, Y -20.970, Z 29.750} C_DIS
   LIN {X -11.926, Y -21.478, Z 29.750} C_DIS
   LIN {X -11.767, Y -24.676, Z 29.750} C_DIS
   LIN {X -10.650, Y -27.143, Z 29.750} C_DIS
   LIN {X -10.544, Y -27.379, Z 29.750} C_DIS
   LIN {X -10.349, Y -27.566, Z 29.750} C_DIS
   LIN {X -7.591, Y -30.132, Z 29.750} C_DIS
   LIN {X -6.359, Y -30.625, Z 29.750} C_DIS
   LIN {X -4.849, Y -31.158, Z 29.750} C_DIS
   LIN {X -3.146, Y -31.232, Z 29.750} C_DIS
   LIN {X -2.198, Y -31.284, Z 29.750} C_DIS
   LIN {X -0.981, Y -30.894, Z 29.750} C_DIS
   LIN {X 1.489, Y -30.072, Z 29.750} C_DIS
   LIN {X 3.434, Y -28.277, Z 29.750} C_DIS
   LIN {X 4.395, Y -27.351, Z 29.750} C_DIS
   LIN {X 5.053, Y -25.902, Z 29.750} C_DIS
   LIN {X 5.672, Y -24.557, Z 29.750} C_DIS
   LIN {X 5.920, Y -23.565, Z 29.750} C_DIS
   LIN {X 6.452, Y -21.389, Z 29.750} C_DIS
   LIN {X 6.961, Y -19.057, Z 29.750} C_DIS
   LIN {X 7.101, Y -18.396, Z 29.750} C_DIS
   LIN {X 7.379, Y -16.867, Z 29.750} C_DIS
   LIN {X 7.806, Y -14.571, Z 29.750} C_DIS
   LIN {X 8.093, Y -12.598, Z 29.750} C_DIS
   LIN {X 8.506, Y -9.679, Z 29.750} C_DIS
   LIN {X 9.032, Y -4.078, Z 29.750}
   LaserEnd_Ext()
   LIN {X -10.280, Y -19.184, Z 29.750}
   LaserStart_Ext()
   LIN {X -10.280, Y -25.536, Z 29.750}
   LaserEnd_Ext()
   LIN {X -9.280, Y -27.195, Z 29.750}
   LaserStart_Ext()
   LIN {X -9.280, Y -17.010, Z 29.750}
   LaserEnd_Ext()
   LIN {X -8.280, Y -15.089, Z 29.750}
   LaserStart_Ext()
   LIN {X -8.280, Y -19.947, Z 29.750}
   LaserEnd_Ext()
   LIN {X -8.280, Y -25.081, Z 29.750}
   LaserStart_Ext()
   LIN {X -8.280, Y -28.125, Z 29.750}
   LaserEnd_Ext()
   LIN {X -7.280, Y -29.055, Z 29.750}
   LaserStart_Ext()
   LIN {X -7.280, Y -26.559, Z 29.750}
   LaserEnd_Ext()
   LIN {X -7.280, Y -18.134, Z 29.750}
   LaserStart_Ext()
   LIN {X -7.280, Y -12.889, Z 29.750}
   LaserEnd_Ext()
   LIN {X -6.280, Y -10.631, Z 29.750}
   LaserStart_Ext()
   LIN {X -6.280, Y -17.398, Z 29.750}
   LaserEnd_Ext()
   LIN {X -6.280, Y -27.278, Z 29.750}
   LaserStart_Ext()
   LIN {X -6.280, Y -29.579, Z 29.750}
   LaserEnd_Ext()
   LIN {X -5.280, Y -29.945, Z 29.750}
   LaserStart_Ext()
   LIN {X -5.280, Y -27.890, Z 29.750}
   LaserEnd_Ext()
   LIN {X -5.280, Y -16.782, Z 29.750}
   LaserStart_Ext()
   LIN {X -5.280, Y -8.030, Z 29.750}
   LaserEnd_Ext()
   LIN {X -4.280, Y -5.079, Z 29.750}
   LaserStart_Ext()
   LIN {X -4.280, Y -16.556, Z 29.750}
   LaserEnd_Ext()
   LIN {X -4.280, Y -28.092, Z 29.750}
   LaserStart_Ext()
   LIN {X -4.280, Y -30.182, Z 29.750}
   LaserEnd_Ext()
   LIN {X -3.280, Y -30.225, Z 29.750}
   LaserStart_Ext()
   LIN {X -3.280, Y -28.295, Z 29.750}
   LaserEnd_Ext()
   LIN {X -3.280, Y -16.329, Z 29.750}
   LaserStart_Ext()
   LIN {X -3.280, Y -1.823, Z 29.750}
   LaserEnd_Ext()
   LIN {X -3.280, Y 36.748, Z 29.750}
   LaserStart_Ext()
   LIN {X -3.280, Y 40.847, Z 29.750}
   LaserEnd_Ext()
   LIN {X -2.280, Y 41.633, Z 29.750}
   LaserStart_Ext()
   LIN {X -2.280, Y 32.533, Z 29.750}
   LaserEnd_Ext()
   LIN {X -2.280, Y 2.755, Z 29.750}
   LaserStart_Ext()
   LIN {X -2.280, Y -16.467, Z 29.750}
   LaserEnd_Ext()
   LIN {X -2.280, Y -28.178, Z 29.750}
   LaserStart_Ext()
   LIN {X -2.280, Y -30.260, Z 29.750}
   LaserEnd_Ext()
   LIN {X -1.280, Y -29.940, Z 29.750}
   LaserStart_Ext()
   LIN {X -1.280, Y -27.959, Z 29.750}
   LaserEnd_Ext()
   LIN {X -1.280, Y -16.658, Z 29.750}
   LaserStart_Ext()
   LIN {X -1.280, Y 8.971, Z 29.750}
   LaserEnd_Ext()
   LIN {X -1.280, Y 26.550, Z 29.750}
   LaserStart_Ext()
   LIN {X -1.280, Y 42.013, Z 29.750}
   LaserEnd_Ext()
   LIN {X -0.280, Y 42.050, Z 29.750}
   LaserStart_Ext()
   LIN {X -0.280, Y -17.033, Z 29.750}
   LaserEnd_Ext()
   LIN {X -0.280, Y -27.591, Z 29.750}
   LaserStart_Ext()
   LIN {X -0.280, Y -29.607, Z 29.750}
   LaserEnd_Ext()
   LIN {X 0.720, Y -29.274, Z 29.750}
   LaserStart_Ext()
   LIN {X 0.720, Y -26.840, Z 29.750}
   LaserEnd_Ext()
   LIN {X 0.720, Y -17.758, Z 29.750}
   LaserStart_Ext()
   LIN {X 0.720, Y 41.631, Z 29.750}
   LaserEnd_Ext()
   LIN {X 1.720, Y 40.556, Z 29.750}
   LaserStart_Ext()
   LIN {X 1.720, Y -18.786, Z 29.750}
   LaserEnd_Ext()
   LIN {X 1.720, Y -25.817, Z 29.750}
   LaserStart_Ext()
   LIN {X 1.720, Y -28.498, Z 29.750}
   LaserEnd_Ext()
   LIN {X 2.720, Y -27.575, Z 29.750}
   LaserStart_Ext()
   LIN {X 2.720, Y -23.869, Z 29.750}
   LaserEnd_Ext()
   LIN {X 2.720, Y -20.743, Z 29.750}
   LaserStart_Ext()
   LIN {X 2.720, Y 37.930, Z 29.750}
   LaserEnd_Ext()
   LIN {X 3.720, Y 34.737, Z 29.750}
   LaserStart_Ext()
   LIN {X 3.720, Y -26.419, Z 29.750}
   LaserEnd_Ext()
   LIN {X 4.720, Y -24.233, Z 29.750}
   LaserStart_Ext()
   LIN {X 4.720, Y 31.170, Z 29.750}
   LaserEnd_Ext()
   LIN {X 5.720, Y 26.763, Z 29.750}
   LaserStart_Ext()
   LIN {X 5.720, Y -20.054, Z 29.750}
   LaserEnd_Ext()
   LIN {X 6.720, Y -14.939, Z 29.750}
   LaserStart_Ext()
   LIN {X 6.720, Y 21.670, Z 29.750}
   LaserEnd_Ext()
   LIN {X 7.720, Y 14.465, Z 29.750}
   LaserStart_Ext()
   LIN {X 7.720, Y -7.351, Z 29.750}
   LaserEnd_Ext()
   LIN {X -6.666, Y -25.670, Z 30.600}
   LaserStart_Ext()
   LIN {X -7.042, Y -25.032, Z 30.600} C_DIS
   LIN {X -7.726, Y -23.878, Z 30.600} C_DIS
   LIN {X -7.879, Y -22.480, Z 30.600} C_DIS
   LIN {X -7.950, Y -21.803, Z 30.600} C_DIS
   LIN {X -7.551, Y -20.903, Z 30.600} C_DIS
   LIN {X -6.705, Y -18.968, Z 30.600} C_DIS
   LIN {X -5.454, Y -18.026, Z 30.600} C_DIS
   LIN {X -5.067, Y -17.740, Z 30.600} C_DIS
   LIN {X -4.765, Y -17.672, Z 30.600} C_DIS
   LIN {X -3.078, Y -17.273, Z 30.600} C_DIS
   LIN {X -1.189, Y -17.630, Z 30.600} C_DIS
   LIN {X -0.966, Y -17.672, Z 30.600} C_DIS
   LIN {X -0.753, Y -17.824, Z 30.600} C_DIS
   LIN {X 0.758, Y -18.913, Z 30.600} C_DIS
   LIN {X 1.790, Y -20.922, Z 30.600} C_DIS
   LIN {X 1.921, Y -21.175, Z 30.600} C_DIS
   LIN {X 1.920, Y -21.392, Z 30.600} C_DIS
   LIN {X 1.910, Y -23.351, Z 30.600} C_DIS
   LIN {X 1.100, Y -24.935, Z 30.600} C_DIS
   LIN {X 0.793, Y -25.544, Z 30.600} C_DIS
   LIN {X 0.253, Y -25.956, Z 30.600} C_DIS
   LIN {X -0.881, Y -26.808, Z 30.600} C_DIS
   LIN {X -2.896, Y -27.263, Z 30.600} C_DIS
   LIN {X -3.022, Y -27.259, Z 30.600} C_DIS
   LIN {X -4.986, Y -26.870, Z 30.600} C_DIS
   LIN {X -6.188, Y -26.014, Z 30.600} C_DIS
   LIN {X -6.666, Y -25.670, Z 30.600}
   LaserEnd_Ext()
   LIN {X -1.901, Y -31.152, Z 30.600}
   LaserStart_Ext()
   LIN {X 1.672, Y -29.962, Z 30.600} C_DIS
   LIN {X 2.468, Y -29.228, Z 30.600} C_DIS
   LIN {X 4.485, Y -27.284, Z 30.600} C_DIS
   LIN {X 5.672, Y -24.669, Z 30.600} C_DIS
   LIN {X 5.753, Y -24.489, Z 30.600} C_DIS
   LIN {X 5.838, Y -24.135, Z 30.600} C_DIS
   LIN {X 6.526, Y -21.319, Z 30.600} C_DIS
   LIN {X 6.807, Y -20.034, Z 30.600} C_DIS
   LIN {X 7.168, Y -18.324, Z 30.600} C_DIS
   LIN {X 7.849, Y -14.578, Z 30.600} C_DIS
   LIN {X 7.880, Y -14.374, Z 30.600} C_DIS
   LIN {X 8.539, Y -9.721, Z 30.600} C_DIS
   LIN {X 8.880, Y -6.086, Z 30.600} C_DIS
   LIN {X 9.068, Y -3.999, Z 30.600} C_DIS
   LIN {X 9.169, Y -2.056, Z 30.600} C_DIS
   LIN {X 9.292, Y 2.795, Z 30.600} C_DIS
   LIN {X 9.166, Y 8.051, Z 30.600} C_DIS
   LIN {X 8.976, Y 12.062, Z 30.600} C_DIS
   LIN {X 8.677, Y 14.934, Z 30.600} C_DIS
   LIN {X 8.004, Y 19.787, Z 30.600} C_DIS
   LIN {X 7.437, Y 23.535, Z 30.600} C_DIS
   LIN {X 7.114, Y 25.018, Z 30.600} C_DIS
   LIN {X 6.569, Y 27.292, Z 30.600} C_DIS
   LIN {X 6.060, Y 29.764, Z 30.600} C_DIS
   LIN {X 5.940, Y 30.327, Z 30.600} C_DIS
   LIN {X 5.881, Y 30.563, Z 30.600} C_DIS
   LIN {X 5.659, Y 31.383, Z 30.600} C_DIS
   LIN {X 5.123, Y 33.382, Z 30.600} C_DIS
   LIN {X 4.938, Y 34.023, Z 30.600} C_DIS
   LIN {X 4.410, Y 35.804, Z 30.600} C_DIS
   LIN {X 4.037, Y 36.984, Z 30.600} C_DIS
   LIN {X 3.732, Y 37.925, Z 30.600} C_DIS
   LIN {X 3.382, Y 38.973, Z 30.600} C_DIS
   LIN {X 2.850, Y 40.499, Z 30.600} C_DIS
   LIN {X 2.816, Y 40.595, Z 30.600} C_DIS
   LIN {X 2.752, Y 40.703, Z 30.600} C_DIS
   LIN {X 2.075, Y 41.866, Z 30.600} C_DIS
   LIN {X 1.075, Y 42.615, Z 30.600} C_DIS
   LIN {X 0.681, Y 42.909, Z 30.600} C_DIS
   LIN {X -0.242, Y 43.099, Z 30.600} C_DIS
   LIN {X -1.029, Y 43.262, Z 30.600} C_DIS
   LIN {X -1.904, Y 42.927, Z 30.600} C_DIS
